(* Logix 5000 project; controller reports 1756-L63 rev 20.11; software revision 20.04; part 10 of 52 *)

        [149].log_data[0].minminute := 45, [149].log_data[0].maxminute := 45, [149].log_data[0].valid := 1, [149].log_data[1].valid := 1, [149].log_data[2].valid := 1, [149].log_data[3].valid := 1, [149].log_data[4].valid := 1, [149].log_data[5].valid := 1, [149].log_data[6].valid := 1, [149].log_data[7].valid := 1, [149].log_data[8].valid := 1, [149].log_data[9].valid := 1, [149].log_data[10].valid := 1, [149].log_data[11].valid := 1, [149].log_data[12].valid := 1, [149].log_data[13].valid := 1, [149].log_data[14].valid := 1, [149].log_data[15].valid := 1, [149].log_data[16].valid := 1, [149].log_data[17].valid := 1, [149].log_data[18].valid := 1, [149].log_data[19].valid := 1, [149].time.Year := 2023, [149].time.Month := 1, [149].time.Day := 18, [149].time.Hour := 12, [149].time.Minute := 49, [149].time.Second := 59, [150].log_data[0].min := 1.0, [150].log_data[0].max := 1.0, [150].log_data[0].total := 300.0, [150].log_data[0].time := 300.0, [150].log_data[0].minminute := 50, [150].log_data[0].maxminute := 50, [150].log_data[0].valid := 1, [150].log_data[1].valid := 1, [150].log_data[2].valid := 1, [150].log_data[3].valid := 1, [150].log_data[4].valid := 1, [150].log_data[5].valid := 1, [150].log_data[6].valid := 1, [150].log_data[7].valid := 1, [150].log_data[8].valid := 1, [150].log_data[9].valid := 1, [150].log_data[10].valid := 1, [150].log_data[11].valid := 1, [150].log_data[12].valid := 1, [150].log_data[13].valid := 1, [150].log_data[14].valid := 1, [150].log_data[15].valid := 1, [150].log_data[16].valid := 1, [150].log_data[17].valid := 1, [150].log_data[18].valid := 1, [150].log_data[19].valid := 1, [150].time.Year := 2023, [150].time.Month := 1, [150].time.Day := 18, [150].time.Hour := 12, [150].time.Minute := 54, [150].time.Second := 59,
        [151].log_data[0].min := 1.0, [151].log_data[0].max := 1.0, [151].log_data[0].total := 300.0, [151].log_data[0].time := 300.0, [151].log_data[0].minminute := 55, [151].log_data[0].maxminute := 55, [151].log_data[0].valid := 1, [151].log_data[1].valid := 1, [151].log_data[2].valid := 1, [151].log_data[3].valid := 1, [151].log_data[4].valid := 1, [151].log_data[5].valid := 1, [151].log_data[6].valid := 1, [151].log_data[7].valid := 1, [151].log_data[8].valid := 1, [151].log_data[9].valid := 1, [151].log_data[10].valid := 1, [151].log_data[11].valid := 1, [151].log_data[12].valid := 1, [151].log_data[13].valid := 1, [151].log_data[14].valid := 1, [151].log_data[15].valid := 1, [151].log_data[16].valid := 1, [151].log_data[17].valid := 1, [151].log_data[18].valid := 1, [151].log_data[19].valid := 1, [151].time.Year := 2023, [151].time.Month := 1, [151].time.Day := 18, [151].time.Hour := 12, [151].time.Minute := 59, [151].time.Second := 59, [152].log_data[0].min := 1.0, [152].log_data[0].max := 1.0, [152].log_data[0].total := 300.0, [152].log_data[0].time := 300.0, [152].log_data[0].valid := 1, [152].log_data[1].valid := 1, [152].log_data[2].valid := 1, [152].log_data[3].valid := 1, [152].log_data[4].valid := 1, [152].log_data[5].valid := 1, [152].log_data[6].valid := 1, [152].log_data[7].valid := 1, [152].log_data[8].valid := 1, [152].log_data[9].valid := 1, [152].log_data[10].valid := 1, [152].log_data[11].valid := 1, [152].log_data[12].valid := 1, [152].log_data[13].valid := 1, [152].log_data[14].valid := 1, [152].log_data[15].valid := 1, [152].log_data[16].valid := 1, [152].log_data[17].valid := 1, [152].log_data[18].valid := 1, [152].log_data[19].valid := 1, [152].time.Year := 2023, [152].time.Month := 1, [152].time.Day := 18, [152].time.Hour := 13,
        [152].time.Minute := 4, [152].time.Second := 59, [153].log_data[0].min := 1.0, [153].log_data[0].max := 1.0, [153].log_data[0].total := 300.0, [153].log_data[0].time := 300.0, [153].log_data[0].minminute := 5, [153].log_data[0].maxminute := 5, [153].log_data[0].valid := 1, [153].log_data[1].valid := 1, [153].log_data[2].valid := 1, [153].log_data[3].valid := 1, [153].log_data[4].valid := 1, [153].log_data[5].valid := 1, [153].log_data[6].valid := 1, [153].log_data[7].valid := 1, [153].log_data[8].valid := 1, [153].log_data[9].valid := 1, [153].log_data[10].valid := 1, [153].log_data[11].valid := 1, [153].log_data[12].valid := 1, [153].log_data[13].valid := 1, [153].log_data[14].valid := 1, [153].log_data[15].valid := 1, [153].log_data[16].valid := 1, [153].log_data[17].valid := 1, [153].log_data[18].valid := 1, [153].log_data[19].valid := 1, [153].time.Year := 2023, [153].time.Month := 1, [153].time.Day := 18, [153].time.Hour := 13, [153].time.Minute := 9, [153].time.Second := 59, [154].log_data[0].min := 1.0, [154].log_data[0].max := 1.0, [154].log_data[0].total := 300.0, [154].log_data[0].time := 300.0, [154].log_data[0].minminute := 10, [154].log_data[0].maxminute := 10, [154].log_data[0].valid := 1, [154].log_data[1].valid := 1, [154].log_data[2].valid := 1, [154].log_data[3].valid := 1, [154].log_data[4].valid := 1, [154].log_data[5].valid := 1, [154].log_data[6].valid := 1, [154].log_data[7].valid := 1, [154].log_data[8].valid := 1, [154].log_data[9].valid := 1, [154].log_data[10].valid := 1, [154].log_data[11].valid := 1, [154].log_data[12].valid := 1, [154].log_data[13].valid := 1, [154].log_data[14].valid := 1, [154].log_data[15].valid := 1, [154].log_data[16].valid := 1, [154].log_data[17].valid := 1, [154].log_data[18].valid := 1, [154].log_data[19].valid := 1,
        [154].time.Year := 2023, [154].time.Month := 1, [154].time.Day := 18, [154].time.Hour := 13, [154].time.Minute := 14, [154].time.Second := 59, [155].log_data[0].min := 1.0, [155].log_data[0].max := 1.0, [155].log_data[0].total := 300.0, [155].log_data[0].time := 300.0, [155].log_data[0].minminute := 15, [155].log_data[0].maxminute := 15, [155].log_data[0].valid := 1, [155].log_data[1].valid := 1, [155].log_data[2].valid := 1, [155].log_data[3].valid := 1, [155].log_data[4].valid := 1, [155].log_data[5].valid := 1, [155].log_data[6].valid := 1, [155].log_data[7].valid := 1, [155].log_data[8].valid := 1, [155].log_data[9].valid := 1, [155].log_data[10].valid := 1, [155].log_data[11].valid := 1, [155].log_data[12].valid := 1, [155].log_data[13].valid := 1, [155].log_data[14].valid := 1, [155].log_data[15].valid := 1, [155].log_data[16].valid := 1, [155].log_data[17].valid := 1, [155].log_data[18].valid := 1, [155].log_data[19].valid := 1, [155].time.Year := 2023, [155].time.Month := 1, [155].time.Day := 18, [155].time.Hour := 13, [155].time.Minute := 19, [155].time.Second := 59, [156].log_data[0].min := 1.0, [156].log_data[0].max := 1.0, [156].log_data[0].total := 300.0, [156].log_data[0].time := 300.0, [156].log_data[0].minminute := 20, [156].log_data[0].maxminute := 20, [156].log_data[0].valid := 1, [156].log_data[1].valid := 1, [156].log_data[2].valid := 1, [156].log_data[3].valid := 1, [156].log_data[4].valid := 1, [156].log_data[5].valid := 1, [156].log_data[6].valid := 1, [156].log_data[7].valid := 1, [156].log_data[8].valid := 1, [156].log_data[9].valid := 1, [156].log_data[10].valid := 1, [156].log_data[11].valid := 1, [156].log_data[12].valid := 1, [156].log_data[13].valid := 1, [156].log_data[14].valid := 1, [156].log_data[15].valid := 1,
        [156].log_data[16].valid := 1, [156].log_data[17].valid := 1, [156].log_data[18].valid := 1, [156].log_data[19].valid := 1, [156].time.Year := 2023, [156].time.Month := 1, [156].time.Day := 18, [156].time.Hour := 13, [156].time.Minute := 24, [156].time.Second := 59, [157].log_data[0].min := 1.0, [157].log_data[0].max := 1.0, [157].log_data[0].total := 300.0, [157].log_data[0].time := 300.0, [157].log_data[0].minminute := 25, [157].log_data[0].maxminute := 25, [157].log_data[0].valid := 1, [157].log_data[1].valid := 1, [157].log_data[2].valid := 1, [157].log_data[3].valid := 1, [157].log_data[4].valid := 1, [157].log_data[5].valid := 1, [157].log_data[6].valid := 1, [157].log_data[7].valid := 1, [157].log_data[8].valid := 1, [157].log_data[9].valid := 1, [157].log_data[10].valid := 1, [157].log_data[11].valid := 1, [157].log_data[12].valid := 1, [157].log_data[13].valid := 1, [157].log_data[14].valid := 1, [157].log_data[15].valid := 1, [157].log_data[16].valid := 1, [157].log_data[17].valid := 1, [157].log_data[18].valid := 1, [157].log_data[19].valid := 1, [157].time.Year := 2023, [157].time.Month := 1, [157].time.Day := 18, [157].time.Hour := 13, [157].time.Minute := 29, [157].time.Second := 59, [158].log_data[0].min := 1.0, [158].log_data[0].max := 1.0, [158].log_data[0].total := 300.0, [158].log_data[0].time := 300.0, [158].log_data[0].minminute := 30, [158].log_data[0].maxminute := 30, [158].log_data[0].valid := 1, [158].log_data[1].valid := 1, [158].log_data[2].valid := 1, [158].log_data[3].valid := 1, [158].log_data[4].valid := 1, [158].log_data[5].valid := 1, [158].log_data[6].valid := 1, [158].log_data[7].valid := 1, [158].log_data[8].valid := 1, [158].log_data[9].valid := 1, [158].log_data[10].valid := 1, [158].log_data[11].valid := 1,
        [158].log_data[12].valid := 1, [158].log_data[13].valid := 1, [158].log_data[14].valid := 1, [158].log_data[15].valid := 1, [158].log_data[16].valid := 1, [158].log_data[17].valid := 1, [158].log_data[18].valid := 1, [158].log_data[19].valid := 1, [158].time.Year := 2023, [158].time.Month := 1, [158].time.Day := 18, [158].time.Hour := 13, [158].time.Minute := 34, [158].time.Second := 59, [159].log_data[0].min := 1.0, [159].log_data[0].max := 1.0, [159].log_data[0].total := 300.0, [159].log_data[0].time := 300.0, [159].log_data[0].minminute := 35, [159].log_data[0].maxminute := 35, [159].log_data[0].valid := 1, [159].log_data[1].valid := 1, [159].log_data[2].valid := 1, [159].log_data[3].valid := 1, [159].log_data[4].valid := 1, [159].log_data[5].valid := 1, [159].log_data[6].valid := 1, [159].log_data[7].valid := 1, [159].log_data[8].valid := 1, [159].log_data[9].valid := 1, [159].log_data[10].valid := 1, [159].log_data[11].valid := 1, [159].log_data[12].valid := 1, [159].log_data[13].valid := 1, [159].log_data[14].valid := 1, [159].log_data[15].valid := 1, [159].log_data[16].valid := 1, [159].log_data[17].valid := 1, [159].log_data[18].valid := 1, [159].log_data[19].valid := 1, [159].time.Year := 2023, [159].time.Month := 1, [159].time.Day := 18, [159].time.Hour := 13, [159].time.Minute := 39, [159].time.Second := 59, [160].log_data[0].min := 1.0, [160].log_data[0].max := 1.0, [160].log_data[0].total := 300.0, [160].log_data[0].time := 300.0, [160].log_data[0].minminute := 40, [160].log_data[0].maxminute := 40, [160].log_data[0].valid := 1, [160].log_data[1].valid := 1, [160].log_data[2].valid := 1, [160].log_data[3].valid := 1, [160].log_data[4].valid := 1, [160].log_data[5].valid := 1, [160].log_data[6].valid := 1, [160].log_data[7].valid := 1,
        [160].log_data[8].valid := 1, [160].log_data[9].valid := 1, [160].log_data[10].valid := 1, [160].log_data[11].valid := 1, [160].log_data[12].valid := 1, [160].log_data[13].valid := 1, [160].log_data[14].valid := 1, [160].log_data[15].valid := 1, [160].log_data[16].valid := 1, [160].log_data[17].valid := 1, [160].log_data[18].valid := 1, [160].log_data[19].valid := 1, [160].time.Year := 2023, [160].time.Month := 1, [160].time.Day := 18, [160].time.Hour := 13, [160].time.Minute := 44, [160].time.Second := 59, [161].log_data[0].min := 1.0, [161].log_data[0].max := 1.0, [161].log_data[0].total := 300.0, [161].log_data[0].time := 300.0, [161].log_data[0].minminute := 45, [161].log_data[0].maxminute := 45, [161].log_data[0].valid := 1, [161].log_data[1].valid := 1, [161].log_data[2].valid := 1, [161].log_data[3].valid := 1, [161].log_data[4].valid := 1, [161].log_data[5].valid := 1, [161].log_data[6].valid := 1, [161].log_data[7].valid := 1, [161].log_data[8].valid := 1, [161].log_data[9].valid := 1, [161].log_data[10].valid := 1, [161].log_data[11].valid := 1, [161].log_data[12].valid := 1, [161].log_data[13].valid := 1, [161].log_data[14].valid := 1, [161].log_data[15].valid := 1, [161].log_data[16].valid := 1, [161].log_data[17].valid := 1, [161].log_data[18].valid := 1, [161].log_data[19].valid := 1, [161].time.Year := 2023, [161].time.Month := 1, [161].time.Day := 18, [161].time.Hour := 13, [161].time.Minute := 49, [161].time.Second := 59, [162].log_data[0].min := 1.0, [162].log_data[0].max := 1.0, [162].log_data[0].total := 300.0, [162].log_data[0].time := 300.0, [162].log_data[0].minminute := 50, [162].log_data[0].maxminute := 50, [162].log_data[0].valid := 1, [162].log_data[1].valid := 1, [162].log_data[2].valid := 1, [162].log_data[3].valid := 1,
        [162].log_data[4].valid := 1, [162].log_data[5].valid := 1, [162].log_data[6].valid := 1, [162].log_data[7].valid := 1, [162].log_data[8].valid := 1, [162].log_data[9].valid := 1, [162].log_data[10].valid := 1, [162].log_data[11].valid := 1, [162].log_data[12].valid := 1, [162].log_data[13].valid := 1, [162].log_data[14].valid := 1, [162].log_data[15].valid := 1, [162].log_data[16].valid := 1, [162].log_data[17].valid := 1, [162].log_data[18].valid := 1, [162].log_data[19].valid := 1, [162].time.Year := 2023, [162].time.Month := 1, [162].time.Day := 18, [162].time.Hour := 13, [162].time.Minute := 54, [162].time.Second := 59, [163].log_data[0].min := 1.0, [163].log_data[0].max := 1.0, [163].log_data[0].total := 300.0, [163].log_data[0].time := 300.0, [163].log_data[0].minminute := 55, [163].log_data[0].maxminute := 55, [163].log_data[0].valid := 1, [163].log_data[1].valid := 1, [163].log_data[2].valid := 1, [163].log_data[3].valid := 1, [163].log_data[4].valid := 1, [163].log_data[5].valid := 1, [163].log_data[6].valid := 1, [163].log_data[7].valid := 1, [163].log_data[8].valid := 1, [163].log_data[9].valid := 1, [163].log_data[10].valid := 1, [163].log_data[11].valid := 1, [163].log_data[12].valid := 1, [163].log_data[13].valid := 1, [163].log_data[14].valid := 1, [163].log_data[15].valid := 1, [163].log_data[16].valid := 1, [163].log_data[17].valid := 1, [163].log_data[18].valid := 1, [163].log_data[19].valid := 1, [163].time.Year := 2023, [163].time.Month := 1, [163].time.Day := 18, [163].time.Hour := 13, [163].time.Minute := 59, [163].time.Second := 59, [164].log_data[0].min := 1.0, [164].log_data[0].max := 1.0, [164].log_data[0].total := 300.0, [164].log_data[0].time := 300.0, [164].log_data[0].valid := 1, [164].log_data[1].valid := 1,
        [164].log_data[2].valid := 1, [164].log_data[3].valid := 1, [164].log_data[4].valid := 1, [164].log_data[5].valid := 1, [164].log_data[6].valid := 1, [164].log_data[7].valid := 1, [164].log_data[8].valid := 1, [164].log_data[9].valid := 1, [164].log_data[10].valid := 1, [164].log_data[11].valid := 1, [164].log_data[12].valid := 1, [164].log_data[13].valid := 1, [164].log_data[14].valid := 1, [164].log_data[15].valid := 1, [164].log_data[16].valid := 1, [164].log_data[17].valid := 1, [164].log_data[18].valid := 1, [164].log_data[19].valid := 1, [164].time.Year := 2023, [164].time.Month := 1, [164].time.Day := 18, [164].time.Hour := 14, [164].time.Minute := 4, [164].time.Second := 59, [165].log_data[0].min := 1.0, [165].log_data[0].max := 1.0, [165].log_data[0].total := 300.0, [165].log_data[0].time := 300.0, [165].log_data[0].minminute := 5, [165].log_data[0].maxminute := 5, [165].log_data[0].valid := 1, [165].log_data[1].valid := 1, [165].log_data[2].valid := 1, [165].log_data[3].valid := 1, [165].log_data[4].valid := 1, [165].log_data[5].valid := 1, [165].log_data[6].valid := 1, [165].log_data[7].valid := 1, [165].log_data[8].valid := 1, [165].log_data[9].valid := 1, [165].log_data[10].valid := 1, [165].log_data[11].valid := 1, [165].log_data[12].valid := 1, [165].log_data[13].valid := 1, [165].log_data[14].valid := 1, [165].log_data[15].valid := 1, [165].log_data[16].valid := 1, [165].log_data[17].valid := 1, [165].log_data[18].valid := 1, [165].log_data[19].valid := 1, [165].time.Year := 2023, [165].time.Month := 1, [165].time.Day := 18, [165].time.Hour := 14, [165].time.Minute := 9, [165].time.Second := 59, [166].log_data[0].min := 1.0, [166].log_data[0].max := 1.0, [166].log_data[0].total := 300.0, [166].log_data[0].time := 300.0,
        [166].log_data[0].minminute := 10, [166].log_data[0].maxminute := 10, [166].log_data[0].valid := 1, [166].log_data[1].valid := 1, [166].log_data[2].valid := 1, [166].log_data[3].valid := 1, [166].log_data[4].valid := 1, [166].log_data[5].valid := 1, [166].log_data[6].valid := 1, [166].log_data[7].valid := 1, [166].log_data[8].valid := 1, [166].log_data[9].valid := 1, [166].log_data[10].valid := 1, [166].log_data[11].valid := 1, [166].log_data[12].valid := 1, [166].log_data[13].valid := 1, [166].log_data[14].valid := 1, [166].log_data[15].valid := 1, [166].log_data[16].valid := 1, [166].log_data[17].valid := 1, [166].log_data[18].valid := 1, [166].log_data[19].valid := 1, [166].time.Year := 2023, [166].time.Month := 1, [166].time.Day := 18, [166].time.Hour := 14, [166].time.Minute := 14, [166].time.Second := 59, [167].log_data[0].min := 1.0, [167].log_data[0].max := 1.0, [167].log_data[0].total := 300.0, [167].log_data[0].time := 300.0, [167].log_data[0].minminute := 15, [167].log_data[0].maxminute := 15, [167].log_data[0].valid := 1, [167].log_data[1].valid := 1, [167].log_data[2].valid := 1, [167].log_data[3].valid := 1, [167].log_data[4].valid := 1, [167].log_data[5].valid := 1, [167].log_data[6].valid := 1, [167].log_data[7].valid := 1, [167].log_data[8].valid := 1, [167].log_data[9].valid := 1, [167].log_data[10].valid := 1, [167].log_data[11].valid := 1, [167].log_data[12].valid := 1, [167].log_data[13].valid := 1, [167].log_data[14].valid := 1, [167].log_data[15].valid := 1, [167].log_data[16].valid := 1, [167].log_data[17].valid := 1, [167].log_data[18].valid := 1, [167].log_data[19].valid := 1, [167].time.Year := 2023, [167].time.Month := 1, [167].time.Day := 18, [167].time.Hour := 14, [167].time.Minute := 19, [167].time.Second := 59,
        [168].log_data[0].min := 1.0, [168].log_data[0].max := 1.0, [168].log_data[0].total := 300.0, [168].log_data[0].time := 300.0, [168].log_data[0].minminute := 20, [168].log_data[0].maxminute := 20, [168].log_data[0].valid := 1, [168].log_data[1].valid := 1, [168].log_data[2].valid := 1, [168].log_data[3].valid := 1, [168].log_data[4].valid := 1, [168].log_data[5].valid := 1, [168].log_data[6].valid := 1, [168].log_data[7].valid := 1, [168].log_data[8].valid := 1, [168].log_data[9].valid := 1, [168].log_data[10].valid := 1, [168].log_data[11].valid := 1, [168].log_data[12].valid := 1, [168].log_data[13].valid := 1, [168].log_data[14].valid := 1, [168].log_data[15].valid := 1, [168].log_data[16].valid := 1, [168].log_data[17].valid := 1, [168].log_data[18].valid := 1, [168].log_data[19].valid := 1, [168].time.Year := 2023, [168].time.Month := 1, [168].time.Day := 18, [168].time.Hour := 14, [168].time.Minute := 24, [168].time.Second := 59, [169].log_data[0].min := 1.0, [169].log_data[0].max := 1.0, [169].log_data[0].total := 300.0, [169].log_data[0].time := 300.0, [169].log_data[0].minminute := 25, [169].log_data[0].maxminute := 25, [169].log_data[0].valid := 1, [169].log_data[1].valid := 1, [169].log_data[2].valid := 1, [169].log_data[3].valid := 1, [169].log_data[4].valid := 1, [169].log_data[5].valid := 1, [169].log_data[6].valid := 1, [169].log_data[7].valid := 1, [169].log_data[8].valid := 1, [169].log_data[9].valid := 1, [169].log_data[10].valid := 1, [169].log_data[11].valid := 1, [169].log_data[12].valid := 1, [169].log_data[13].valid := 1, [169].log_data[14].valid := 1, [169].log_data[15].valid := 1, [169].log_data[16].valid := 1, [169].log_data[17].valid := 1, [169].log_data[18].valid := 1, [169].log_data[19].valid := 1, [169].time.Year := 2023, [169].time.Month := 1,
        [169].time.Day := 18, [169].time.Hour := 14, [169].time.Minute := 29, [169].time.Second := 59, [170].log_data[0].min := 1.0, [170].log_data[0].max := 1.0, [170].log_data[0].total := 300.0, [170].log_data[0].time := 300.0, [170].log_data[0].minminute := 30, [170].log_data[0].maxminute := 30, [170].log_data[0].valid := 1, [170].log_data[1].valid := 1, [170].log_data[2].valid := 1, [170].log_data[3].valid := 1, [170].log_data[4].valid := 1, [170].log_data[5].valid := 1, [170].log_data[6].valid := 1, [170].log_data[7].valid := 1, [170].log_data[8].valid := 1, [170].log_data[9].valid := 1, [170].log_data[10].valid := 1, [170].log_data[11].valid := 1, [170].log_data[12].valid := 1, [170].log_data[13].valid := 1, [170].log_data[14].valid := 1, [170].log_data[15].valid := 1, [170].log_data[16].valid := 1, [170].log_data[17].valid := 1, [170].log_data[18].valid := 1, [170].log_data[19].valid := 1, [170].time.Year := 2023, [170].time.Month := 1, [170].time.Day := 18, [170].time.Hour := 14, [170].time.Minute := 34, [170].time.Second := 59, [171].log_data[0].min := 1.0, [171].log_data[0].max := 1.0, [171].log_data[0].total := 300.0, [171].log_data[0].time := 300.0, [171].log_data[0].minminute := 35, [171].log_data[0].maxminute := 35, [171].log_data[0].valid := 1, [171].log_data[1].valid := 1, [171].log_data[2].valid := 1, [171].log_data[3].valid := 1, [171].log_data[4].valid := 1, [171].log_data[5].valid := 1, [171].log_data[6].valid := 1, [171].log_data[7].valid := 1, [171].log_data[8].valid := 1, [171].log_data[9].valid := 1, [171].log_data[10].valid := 1, [171].log_data[11].valid := 1, [171].log_data[12].valid := 1, [171].log_data[13].valid := 1, [171].log_data[14].valid := 1, [171].log_data[15].valid := 1, [171].log_data[16].valid := 1, [171].log_data[17].valid := 1,
        [171].log_data[18].valid := 1, [171].log_data[19].valid := 1, [171].time.Year := 2023, [171].time.Month := 1, [171].time.Day := 18, [171].time.Hour := 14, [171].time.Minute := 39, [171].time.Second := 59, [172].log_data[0].min := 1.0, [172].log_data[0].max := 1.0, [172].log_data[0].total := 300.0, [172].log_data[0].time := 300.0, [172].log_data[0].minminute := 40, [172].log_data[0].maxminute := 40, [172].log_data[0].valid := 1, [172].log_data[1].valid := 1, [172].log_data[2].valid := 1, [172].log_data[3].valid := 1, [172].log_data[4].valid := 1, [172].log_data[5].valid := 1, [172].log_data[6].valid := 1, [172].log_data[7].valid := 1, [172].log_data[8].valid := 1, [172].log_data[9].valid := 1, [172].log_data[10].valid := 1, [172].log_data[11].valid := 1, [172].log_data[12].valid := 1, [172].log_data[13].valid := 1, [172].log_data[14].valid := 1, [172].log_data[15].valid := 1, [172].log_data[16].valid := 1, [172].log_data[17].valid := 1, [172].log_data[18].valid := 1, [172].log_data[19].valid := 1, [172].time.Year := 2023, [172].time.Month := 1, [172].time.Day := 18, [172].time.Hour := 14, [172].time.Minute := 44, [172].time.Second := 59, [173].log_data[0].min := 1.0, [173].log_data[0].max := 1.0, [173].log_data[0].total := 300.0, [173].log_data[0].time := 300.0, [173].log_data[0].minminute := 45, [173].log_data[0].maxminute := 45, [173].log_data[0].valid := 1, [173].log_data[1].valid := 1, [173].log_data[2].valid := 1, [173].log_data[3].valid := 1, [173].log_data[4].valid := 1, [173].log_data[5].valid := 1, [173].log_data[6].valid := 1, [173].log_data[7].valid := 1, [173].log_data[8].valid := 1, [173].log_data[9].valid := 1, [173].log_data[10].valid := 1, [173].log_data[11].valid := 1, [173].log_data[12].valid := 1, [173].log_data[13].valid := 1,
        [173].log_data[14].valid := 1, [173].log_data[15].valid := 1, [173].log_data[16].valid := 1, [173].log_data[17].valid := 1, [173].log_data[18].valid := 1, [173].log_data[19].valid := 1, [173].time.Year := 2023, [173].time.Month := 1, [173].time.Day := 18, [173].time.Hour := 14, [173].time.Minute := 49, [173].time.Second := 59, [174].log_data[0].min := 1.0, [174].log_data[0].max := 1.0, [174].log_data[0].total := 300.0, [174].log_data[0].time := 300.0, [174].log_data[0].minminute := 50, [174].log_data[0].maxminute := 50, [174].log_data[0].valid := 1, [174].log_data[1].valid := 1, [174].log_data[2].valid := 1, [174].log_data[3].valid := 1, [174].log_data[4].valid := 1, [174].log_data[5].valid := 1, [174].log_data[6].valid := 1, [174].log_data[7].valid := 1, [174].log_data[8].valid := 1, [174].log_data[9].valid := 1, [174].log_data[10].valid := 1, [174].log_data[11].valid := 1, [174].log_data[12].valid := 1, [174].log_data[13].valid := 1, [174].log_data[14].valid := 1, [174].log_data[15].valid := 1, [174].log_data[16].valid := 1, [174].log_data[17].valid := 1, [174].log_data[18].valid := 1, [174].log_data[19].valid := 1, [174].time.Year := 2023, [174].time.Month := 1, [174].time.Day := 18, [174].time.Hour := 14, [174].time.Minute := 54, [174].time.Second := 59, [175].log_data[0].min := 1.0, [175].log_data[0].max := 1.0, [175].log_data[0].total := 300.0, [175].log_data[0].time := 300.0, [175].log_data[0].minminute := 55, [175].log_data[0].maxminute := 55, [175].log_data[0].valid := 1, [175].log_data[1].valid := 1, [175].log_data[2].valid := 1, [175].log_data[3].valid := 1, [175].log_data[4].valid := 1, [175].log_data[5].valid := 1, [175].log_data[6].valid := 1, [175].log_data[7].valid := 1, [175].log_data[8].valid := 1, [175].log_data[9].valid := 1,
        [175].log_data[10].valid := 1, [175].log_data[11].valid := 1, [175].log_data[12].valid := 1, [175].log_data[13].valid := 1, [175].log_data[14].valid := 1, [175].log_data[15].valid := 1, [175].log_data[16].valid := 1, [175].log_data[17].valid := 1, [175].log_data[18].valid := 1, [175].log_data[19].valid := 1, [175].time.Year := 2023, [175].time.Month := 1, [175].time.Day := 18, [175].time.Hour := 14, [175].time.Minute := 59, [175].time.Second := 59, [176].log_data[0].min := 1.0, [176].log_data[0].max := 1.0, [176].log_data[0].total := 300.0, [176].log_data[0].time := 300.0, [176].log_data[0].valid := 1, [176].log_data[1].valid := 1, [176].log_data[2].valid := 1, [176].log_data[3].valid := 1, [176].log_data[4].valid := 1, [176].log_data[5].valid := 1, [176].log_data[6].valid := 1, [176].log_data[7].valid := 1, [176].log_data[8].valid := 1, [176].log_data[9].valid := 1, [176].log_data[10].valid := 1, [176].log_data[11].valid := 1, [176].log_data[12].valid := 1, [176].log_data[13].valid := 1, [176].log_data[14].valid := 1, [176].log_data[15].valid := 1, [176].log_data[16].valid := 1, [176].log_data[17].valid := 1, [176].log_data[18].valid := 1, [176].log_data[19].valid := 1, [176].time.Year := 2023, [176].time.Month := 1, [176].time.Day := 18, [176].time.Hour := 15, [176].time.Minute := 4, [176].time.Second := 59, [177].log_data[0].min := 1.0, [177].log_data[0].max := 1.0, [177].log_data[0].total := 300.0, [177].log_data[0].time := 300.0, [177].log_data[0].minminute := 5, [177].log_data[0].maxminute := 5, [177].log_data[0].valid := 1, [177].log_data[1].valid := 1, [177].log_data[2].valid := 1, [177].log_data[3].valid := 1, [177].log_data[4].valid := 1, [177].log_data[5].valid := 1, [177].log_data[6].valid := 1, [177].log_data[7].valid := 1,
        [177].log_data[8].valid := 1, [177].log_data[9].valid := 1, [177].log_data[10].valid := 1, [177].log_data[11].valid := 1, [177].log_data[12].valid := 1, [177].log_data[13].valid := 1, [177].log_data[14].valid := 1, [177].log_data[15].valid := 1, [177].log_data[16].valid := 1, [177].log_data[17].valid := 1, [177].log_data[18].valid := 1, [177].log_data[19].valid := 1, [177].time.Year := 2023, [177].time.Month := 1, [177].time.Day := 18, [177].time.Hour := 15, [177].time.Minute := 9, [177].time.Second := 59, [178].log_data[0].min := 1.0, [178].log_data[0].max := 1.0, [178].log_data[0].total := 300.0, [178].log_data[0].time := 300.0, [178].log_data[0].minminute := 10, [178].log_data[0].maxminute := 10, [178].log_data[0].valid := 1, [178].log_data[1].valid := 1, [178].log_data[2].valid := 1, [178].log_data[3].valid := 1, [178].log_data[4].valid := 1, [178].log_data[5].valid := 1, [178].log_data[6].valid := 1, [178].log_data[7].valid := 1, [178].log_data[8].valid := 1, [178].log_data[9].valid := 1, [178].log_data[10].valid := 1, [178].log_data[11].valid := 1, [178].log_data[12].valid := 1, [178].log_data[13].valid := 1, [178].log_data[14].valid := 1, [178].log_data[15].valid := 1, [178].log_data[16].valid := 1, [178].log_data[17].valid := 1, [178].log_data[18].valid := 1, [178].log_data[19].valid := 1, [178].time.Year := 2023, [178].time.Month := 1, [178].time.Day := 18, [178].time.Hour := 15, [178].time.Minute := 14, [178].time.Second := 59, [179].log_data[0].min := 1.0, [179].log_data[0].max := 1.0, [179].log_data[0].total := 300.0, [179].log_data[0].time := 300.0, [179].log_data[0].minminute := 15, [179].log_data[0].maxminute := 15, [179].log_data[0].valid := 1, [179].log_data[1].valid := 1, [179].log_data[2].valid := 1, [179].log_data[3].valid := 1,
        [179].log_data[4].valid := 1, [179].log_data[5].valid := 1, [179].log_data[6].valid := 1, [179].log_data[7].valid := 1, [179].log_data[8].valid := 1, [179].log_data[9].valid := 1, [179].log_data[10].valid := 1, [179].log_data[11].valid := 1, [179].log_data[12].valid := 1, [179].log_data[13].valid := 1, [179].log_data[14].valid := 1, [179].log_data[15].valid := 1, [179].log_data[16].valid := 1, [179].log_data[17].valid := 1, [179].log_data[18].valid := 1, [179].log_data[19].valid := 1, [179].time.Year := 2023, [179].time.Month := 1, [179].time.Day := 18, [179].time.Hour := 15, [179].time.Minute := 19, [179].time.Second := 59, [180].log_data[0].min := 1.0, [180].log_data[0].max := 1.0, [180].log_data[0].total := 300.0, [180].log_data[0].time := 300.0, [180].log_data[0].minminute := 20, [180].log_data[0].maxminute := 20, [180].log_data[0].valid := 1, [180].log_data[1].valid := 1, [180].log_data[2].valid := 1, [180].log_data[3].valid := 1, [180].log_data[4].valid := 1, [180].log_data[5].valid := 1, [180].log_data[6].valid := 1, [180].log_data[7].valid := 1, [180].log_data[8].valid := 1, [180].log_data[9].valid := 1, [180].log_data[10].valid := 1, [180].log_data[11].valid := 1, [180].log_data[12].valid := 1, [180].log_data[13].valid := 1, [180].log_data[14].valid := 1, [180].log_data[15].valid := 1, [180].log_data[16].valid := 1, [180].log_data[17].valid := 1, [180].log_data[18].valid := 1, [180].log_data[19].valid := 1, [180].time.Year := 2023, [180].time.Month := 1, [180].time.Day := 18, [180].time.Hour := 15, [180].time.Minute := 24, [180].time.Second := 59, [181].log_data[0].min := 1.0, [181].log_data[0].max := 1.0, [181].log_data[0].total := 300.0, [181].log_data[0].time := 300.0, [181].log_data[0].minminute := 25, [181].log_data[0].maxminute := 25,
        [181].log_data[0].valid := 1, [181].log_data[1].valid := 1, [181].log_data[2].valid := 1, [181].log_data[3].valid := 1, [181].log_data[4].valid := 1, [181].log_data[5].valid := 1, [181].log_data[6].valid := 1, [181].log_data[7].valid := 1, [181].log_data[8].valid := 1, [181].log_data[9].valid := 1, [181].log_data[10].valid := 1, [181].log_data[11].valid := 1, [181].log_data[12].valid := 1, [181].log_data[13].valid := 1, [181].log_data[14].valid := 1, [181].log_data[15].valid := 1, [181].log_data[16].valid := 1, [181].log_data[17].valid := 1, [181].log_data[18].valid := 1, [181].log_data[19].valid := 1, [181].time.Year := 2023, [181].time.Month := 1, [181].time.Day := 18, [181].time.Hour := 15, [181].time.Minute := 29, [181].time.Second := 59, [182].log_data[0].min := 1.0, [182].log_data[0].max := 1.0, [182].log_data[0].total := 300.0, [182].log_data[0].time := 300.0, [182].log_data[0].minminute := 30, [182].log_data[0].maxminute := 30, [182].log_data[0].valid := 1, [182].log_data[1].valid := 1, [182].log_data[2].valid := 1, [182].log_data[3].valid := 1, [182].log_data[4].valid := 1, [182].log_data[5].valid := 1, [182].log_data[6].valid := 1, [182].log_data[7].valid := 1, [182].log_data[8].valid := 1, [182].log_data[9].valid := 1, [182].log_data[10].valid := 1, [182].log_data[11].valid := 1, [182].log_data[12].valid := 1, [182].log_data[13].valid := 1, [182].log_data[14].valid := 1, [182].log_data[15].valid := 1, [182].log_data[16].valid := 1, [182].log_data[17].valid := 1, [182].log_data[18].valid := 1, [182].log_data[19].valid := 1, [182].time.Year := 2023, [182].time.Month := 1, [182].time.Day := 18, [182].time.Hour := 15, [182].time.Minute := 34, [182].time.Second := 59, [183].log_data[0].min := 1.0, [183].log_data[0].max := 1.0,
        [183].log_data[0].total := 300.0, [183].log_data[0].time := 300.0, [183].log_data[0].minminute := 35, [183].log_data[0].maxminute := 35, [183].log_data[0].valid := 1, [183].log_data[1].valid := 1, [183].log_data[2].valid := 1, [183].log_data[3].valid := 1, [183].log_data[4].valid := 1, [183].log_data[5].valid := 1, [183].log_data[6].valid := 1, [183].log_data[7].valid := 1, [183].log_data[8].valid := 1, [183].log_data[9].valid := 1, [183].log_data[10].valid := 1, [183].log_data[11].valid := 1, [183].log_data[12].valid := 1, [183].log_data[13].valid := 1, [183].log_data[14].valid := 1, [183].log_data[15].valid := 1, [183].log_data[16].valid := 1, [183].log_data[17].valid := 1, [183].log_data[18].valid := 1, [183].log_data[19].valid := 1, [183].time.Year := 2023, [183].time.Month := 1, [183].time.Day := 18, [183].time.Hour := 15, [183].time.Minute := 39, [183].time.Second := 59, [184].log_data[0].min := 1.0, [184].log_data[0].max := 1.0, [184].log_data[0].total := 300.0, [184].log_data[0].time := 300.0, [184].log_data[0].minminute := 40, [184].log_data[0].maxminute := 40, [184].log_data[0].valid := 1, [184].log_data[1].valid := 1, [184].log_data[2].valid := 1, [184].log_data[3].valid := 1, [184].log_data[4].valid := 1, [184].log_data[5].valid := 1, [184].log_data[6].valid := 1, [184].log_data[7].valid := 1, [184].log_data[8].valid := 1, [184].log_data[9].valid := 1, [184].log_data[10].valid := 1, [184].log_data[11].valid := 1, [184].log_data[12].valid := 1, [184].log_data[13].valid := 1, [184].log_data[14].valid := 1, [184].log_data[15].valid := 1, [184].log_data[16].valid := 1, [184].log_data[17].valid := 1, [184].log_data[18].valid := 1, [184].log_data[19].valid := 1, [184].time.Year := 2023, [184].time.Month := 1, [184].time.Day := 18, [184].time.Hour := 15,
        [184].time.Minute := 44, [184].time.Second := 59, [185].log_data[0].min := 1.0, [185].log_data[0].max := 1.0, [185].log_data[0].total := 300.0, [185].log_data[0].time := 300.0, [185].log_data[0].minminute := 45, [185].log_data[0].maxminute := 45, [185].log_data[0].valid := 1, [185].log_data[1].valid := 1, [185].log_data[2].valid := 1, [185].log_data[3].valid := 1, [185].log_data[4].valid := 1, [185].log_data[5].valid := 1, [185].log_data[6].valid := 1, [185].log_data[7].valid := 1, [185].log_data[8].valid := 1, [185].log_data[9].valid := 1, [185].log_data[10].valid := 1, [185].log_data[11].valid := 1, [185].log_data[12].valid := 1, [185].log_data[13].valid := 1, [185].log_data[14].valid := 1, [185].log_data[15].valid := 1, [185].log_data[16].valid := 1, [185].log_data[17].valid := 1, [185].log_data[18].valid := 1, [185].log_data[19].valid := 1, [185].time.Year := 2023, [185].time.Month := 1, [185].time.Day := 18, [185].time.Hour := 15, [185].time.Minute := 49, [185].time.Second := 59, [186].log_data[0].min := 1.0, [186].log_data[0].max := 1.0, [186].log_data[0].total := 300.0, [186].log_data[0].time := 300.0, [186].log_data[0].minminute := 50, [186].log_data[0].maxminute := 50, [186].log_data[0].valid := 1, [186].log_data[1].valid := 1, [186].log_data[2].valid := 1, [186].log_data[3].valid := 1, [186].log_data[4].valid := 1, [186].log_data[5].valid := 1, [186].log_data[6].valid := 1, [186].log_data[7].valid := 1, [186].log_data[8].valid := 1, [186].log_data[9].valid := 1, [186].log_data[10].valid := 1, [186].log_data[11].valid := 1, [186].log_data[12].valid := 1, [186].log_data[13].valid := 1, [186].log_data[14].valid := 1, [186].log_data[15].valid := 1, [186].log_data[16].valid := 1, [186].log_data[17].valid := 1, [186].log_data[18].valid := 1, [186].log_data[19].valid := 1,
        [186].time.Year := 2023, [186].time.Month := 1, [186].time.Day := 18, [186].time.Hour := 15, [186].time.Minute := 54, [186].time.Second := 59, [187].log_data[0].min := 1.0, [187].log_data[0].max := 1.0, [187].log_data[0].total := 300.0, [187].log_data[0].time := 300.0, [187].log_data[0].minminute := 55, [187].log_data[0].maxminute := 55, [187].log_data[0].valid := 1, [187].log_data[1].valid := 1, [187].log_data[2].valid := 1, [187].log_data[3].valid := 1, [187].log_data[4].valid := 1, [187].log_data[5].valid := 1, [187].log_data[6].valid := 1, [187].log_data[7].valid := 1, [187].log_data[8].valid := 1, [187].log_data[9].valid := 1, [187].log_data[10].valid := 1, [187].log_data[11].valid := 1, [187].log_data[12].valid := 1, [187].log_data[13].valid := 1, [187].log_data[14].valid := 1, [187].log_data[15].valid := 1, [187].log_data[16].valid := 1, [187].log_data[17].valid := 1, [187].log_data[18].valid := 1, [187].log_data[19].valid := 1, [187].time.Year := 2023, [187].time.Month := 1, [187].time.Day := 18, [187].time.Hour := 15, [187].time.Minute := 59, [187].time.Second := 59, [188].log_data[0].min := 1.0, [188].log_data[0].max := 1.0, [188].log_data[0].total := 300.0, [188].log_data[0].time := 300.0, [188].log_data[0].valid := 1, [188].log_data[1].valid := 1, [188].log_data[2].valid := 1, [188].log_data[3].valid := 1, [188].log_data[4].valid := 1, [188].log_data[5].valid := 1, [188].log_data[6].valid := 1, [188].log_data[7].valid := 1, [188].log_data[8].valid := 1, [188].log_data[9].valid := 1, [188].log_data[10].valid := 1, [188].log_data[11].valid := 1, [188].log_data[12].valid := 1, [188].log_data[13].valid := 1, [188].log_data[14].valid := 1, [188].log_data[15].valid := 1, [188].log_data[16].valid := 1, [188].log_data[17].valid := 1,
        [188].log_data[18].valid := 1, [188].log_data[19].valid := 1, [188].time.Year := 2023, [188].time.Month := 1, [188].time.Day := 18, [188].time.Hour := 16, [188].time.Minute := 4, [188].time.Second := 59, [189].log_data[0].min := 1.0, [189].log_data[0].max := 1.0, [189].log_data[0].total := 300.0, [189].log_data[0].time := 300.0, [189].log_data[0].minminute := 5, [189].log_data[0].maxminute := 5, [189].log_data[0].valid := 1, [189].log_data[1].valid := 1, [189].log_data[2].valid := 1, [189].log_data[3].valid := 1, [189].log_data[4].valid := 1, [189].log_data[5].valid := 1, [189].log_data[6].valid := 1, [189].log_data[7].valid := 1, [189].log_data[8].valid := 1, [189].log_data[9].valid := 1, [189].log_data[10].valid := 1, [189].log_data[11].valid := 1, [189].log_data[12].valid := 1, [189].log_data[13].valid := 1, [189].log_data[14].valid := 1, [189].log_data[15].valid := 1, [189].log_data[16].valid := 1, [189].log_data[17].valid := 1, [189].log_data[18].valid := 1, [189].log_data[19].valid := 1, [189].time.Year := 2023, [189].time.Month := 1, [189].time.Day := 18, [189].time.Hour := 16, [189].time.Minute := 9, [189].time.Second := 59, [190].log_data[0].min := 1.0, [190].log_data[0].max := 1.0, [190].log_data[0].total := 300.0, [190].log_data[0].time := 300.0, [190].log_data[0].minminute := 10, [190].log_data[0].maxminute := 10, [190].log_data[0].valid := 1, [190].log_data[1].valid := 1, [190].log_data[2].valid := 1, [190].log_data[3].valid := 1, [190].log_data[4].valid := 1, [190].log_data[5].valid := 1, [190].log_data[6].valid := 1, [190].log_data[7].valid := 1, [190].log_data[8].valid := 1, [190].log_data[9].valid := 1, [190].log_data[10].valid := 1, [190].log_data[11].valid := 1, [190].log_data[12].valid := 1, [190].log_data[13].valid := 1,
        [190].log_data[14].valid := 1, [190].log_data[15].valid := 1, [190].log_data[16].valid := 1, [190].log_data[17].valid := 1, [190].log_data[18].valid := 1, [190].log_data[19].valid := 1, [190].time.Year := 2023, [190].time.Month := 1, [190].time.Day := 18, [190].time.Hour := 16, [190].time.Minute := 14, [190].time.Second := 59, [191].log_data[0].min := 1.0, [191].log_data[0].max := 1.0, [191].log_data[0].total := 300.0, [191].log_data[0].time := 300.0, [191].log_data[0].minminute := 15, [191].log_data[0].maxminute := 15, [191].log_data[0].valid := 1, [191].log_data[1].valid := 1, [191].log_data[2].valid := 1, [191].log_data[3].valid := 1, [191].log_data[4].valid := 1, [191].log_data[5].valid := 1, [191].log_data[6].valid := 1, [191].log_data[7].valid := 1, [191].log_data[8].valid := 1, [191].log_data[9].valid := 1, [191].log_data[10].valid := 1, [191].log_data[11].valid := 1, [191].log_data[12].valid := 1, [191].log_data[13].valid := 1, [191].log_data[14].valid := 1, [191].log_data[15].valid := 1, [191].log_data[16].valid := 1, [191].log_data[17].valid := 1, [191].log_data[18].valid := 1, [191].log_data[19].valid := 1, [191].time.Year := 2023, [191].time.Month := 1, [191].time.Day := 18, [191].time.Hour := 16, [191].time.Minute := 19, [191].time.Second := 59, [192].log_data[0].min := 1.0, [192].log_data[0].max := 1.0, [192].log_data[0].total := 300.0, [192].log_data[0].time := 300.0, [192].log_data[0].minminute := 20, [192].log_data[0].maxminute := 20, [192].log_data[0].valid := 1, [192].log_data[1].valid := 1, [192].log_data[2].valid := 1, [192].log_data[3].valid := 1, [192].log_data[4].valid := 1, [192].log_data[5].valid := 1, [192].log_data[6].valid := 1, [192].log_data[7].valid := 1, [192].log_data[8].valid := 1, [192].log_data[9].valid := 1,
        [192].log_data[10].valid := 1, [192].log_data[11].valid := 1, [192].log_data[12].valid := 1, [192].log_data[13].valid := 1, [192].log_data[14].valid := 1, [192].log_data[15].valid := 1, [192].log_data[16].valid := 1, [192].log_data[17].valid := 1, [192].log_data[18].valid := 1, [192].log_data[19].valid := 1, [192].time.Year := 2023, [192].time.Month := 1, [192].time.Day := 18, [192].time.Hour := 16, [192].time.Minute := 24, [192].time.Second := 59, [193].log_data[0].min := 1.0, [193].log_data[0].max := 1.0, [193].log_data[0].total := 300.0, [193].log_data[0].time := 300.0, [193].log_data[0].minminute := 25, [193].log_data[0].maxminute := 25, [193].log_data[0].valid := 1, [193].log_data[1].valid := 1, [193].log_data[2].valid := 1, [193].log_data[3].valid := 1, [193].log_data[4].valid := 1, [193].log_data[5].valid := 1, [193].log_data[6].valid := 1, [193].log_data[7].valid := 1, [193].log_data[8].valid := 1, [193].log_data[9].valid := 1, [193].log_data[10].valid := 1, [193].log_data[11].valid := 1, [193].log_data[12].valid := 1, [193].log_data[13].valid := 1, [193].log_data[14].valid := 1, [193].log_data[15].valid := 1, [193].log_data[16].valid := 1, [193].log_data[17].valid := 1, [193].log_data[18].valid := 1, [193].log_data[19].valid := 1, [193].time.Year := 2023, [193].time.Month := 1, [193].time.Day := 18, [193].time.Hour := 16, [193].time.Minute := 29, [193].time.Second := 59, [194].log_data[0].min := 1.0, [194].log_data[0].max := 1.0, [194].log_data[0].total := 300.0, [194].log_data[0].time := 300.0, [194].log_data[0].minminute := 30, [194].log_data[0].maxminute := 30, [194].log_data[0].valid := 1, [194].log_data[1].valid := 1, [194].log_data[2].valid := 1, [194].log_data[3].valid := 1, [194].log_data[4].valid := 1, [194].log_data[5].valid := 1,
        [194].log_data[6].valid := 1, [194].log_data[7].valid := 1, [194].log_data[8].valid := 1, [194].log_data[9].valid := 1, [194].log_data[10].valid := 1, [194].log_data[11].valid := 1, [194].log_data[12].valid := 1, [194].log_data[13].valid := 1, [194].log_data[14].valid := 1, [194].log_data[15].valid := 1, [194].log_data[16].valid := 1, [194].log_data[17].valid := 1, [194].log_data[18].valid := 1, [194].log_data[19].valid := 1, [194].time.Year := 2023, [194].time.Month := 1, [194].time.Day := 18, [194].time.Hour := 16, [194].time.Minute := 34, [194].time.Second := 59, [195].log_data[0].min := 1.0, [195].log_data[0].max := 1.0, [195].log_data[0].total := 300.0, [195].log_data[0].time := 300.0, [195].log_data[0].minminute := 35, [195].log_data[0].maxminute := 35, [195].log_data[0].valid := 1, [195].log_data[1].valid := 1, [195].log_data[2].valid := 1, [195].log_data[3].valid := 1, [195].log_data[4].valid := 1, [195].log_data[5].valid := 1, [195].log_data[6].valid := 1, [195].log_data[7].valid := 1, [195].log_data[8].valid := 1, [195].log_data[9].valid := 1, [195].log_data[10].valid := 1, [195].log_data[11].valid := 1, [195].log_data[12].valid := 1, [195].log_data[13].valid := 1, [195].log_data[14].valid := 1, [195].log_data[15].valid := 1, [195].log_data[16].valid := 1, [195].log_data[17].valid := 1, [195].log_data[18].valid := 1, [195].log_data[19].valid := 1, [195].time.Year := 2023, [195].time.Month := 1, [195].time.Day := 18, [195].time.Hour := 16, [195].time.Minute := 39, [195].time.Second := 59, [196].log_data[0].min := 1.0, [196].log_data[0].max := 1.0, [196].log_data[0].total := 300.0, [196].log_data[0].time := 300.0, [196].log_data[0].minminute := 40, [196].log_data[0].maxminute := 40, [196].log_data[0].valid := 1, [196].log_data[1].valid := 1,
        [196].log_data[2].valid := 1, [196].log_data[3].valid := 1, [196].log_data[4].valid := 1, [196].log_data[5].valid := 1, [196].log_data[6].valid := 1, [196].log_data[7].valid := 1, [196].log_data[8].valid := 1, [196].log_data[9].valid := 1, [196].log_data[10].valid := 1, [196].log_data[11].valid := 1, [196].log_data[12].valid := 1, [196].log_data[13].valid := 1, [196].log_data[14].valid := 1, [196].log_data[15].valid := 1, [196].log_data[16].valid := 1, [196].log_data[17].valid := 1, [196].log_data[18].valid := 1, [196].log_data[19].valid := 1, [196].time.Year := 2023, [196].time.Month := 1, [196].time.Day := 18, [196].time.Hour := 16, [196].time.Minute := 44, [196].time.Second := 59, [197].log_data[0].min := 1.0, [197].log_data[0].max := 1.0, [197].log_data[0].total := 300.0, [197].log_data[0].time := 300.0, [197].log_data[0].minminute := 45, [197].log_data[0].maxminute := 45, [197].log_data[0].valid := 1, [197].log_data[1].valid := 1, [197].log_data[2].valid := 1, [197].log_data[3].valid := 1, [197].log_data[4].valid := 1, [197].log_data[5].valid := 1, [197].log_data[6].valid := 1, [197].log_data[7].valid := 1, [197].log_data[8].valid := 1, [197].log_data[9].valid := 1, [197].log_data[10].valid := 1, [197].log_data[11].valid := 1, [197].log_data[12].valid := 1, [197].log_data[13].valid := 1, [197].log_data[14].valid := 1, [197].log_data[15].valid := 1, [197].log_data[16].valid := 1, [197].log_data[17].valid := 1, [197].log_data[18].valid := 1, [197].log_data[19].valid := 1, [197].time.Year := 2023, [197].time.Month := 1, [197].time.Day := 18, [197].time.Hour := 16, [197].time.Minute := 49, [197].time.Second := 59, [198].log_data[0].min := 1.0, [198].log_data[0].max := 1.0, [198].log_data[0].total := 300.0, [198].log_data[0].time := 300.0,
        [198].log_data[0].minminute := 50, [198].log_data[0].maxminute := 50, [198].log_data[0].valid := 1, [198].log_data[1].valid := 1, [198].log_data[2].valid := 1, [198].log_data[3].valid := 1, [198].log_data[4].valid := 1, [198].log_data[5].valid := 1, [198].log_data[6].valid := 1, [198].log_data[7].valid := 1, [198].log_data[8].valid := 1, [198].log_data[9].valid := 1, [198].log_data[10].valid := 1, [198].log_data[11].valid := 1, [198].log_data[12].valid := 1, [198].log_data[13].valid := 1, [198].log_data[14].valid := 1, [198].log_data[15].valid := 1, [198].log_data[16].valid := 1, [198].log_data[17].valid := 1, [198].log_data[18].valid := 1, [198].log_data[19].valid := 1, [198].time.Year := 2023, [198].time.Month := 1, [198].time.Day := 18, [198].time.Hour := 16, [198].time.Minute := 54, [198].time.Second := 59, [199].log_data[0].min := 1.0, [199].log_data[0].max := 1.0, [199].log_data[0].total := 300.0, [199].log_data[0].time := 300.0, [199].log_data[0].minminute := 55, [199].log_data[0].maxminute := 55, [199].log_data[0].valid := 1, [199].log_data[1].valid := 1, [199].log_data[2].valid := 1, [199].log_data[3].valid := 1, [199].log_data[4].valid := 1, [199].log_data[5].valid := 1, [199].log_data[6].valid := 1, [199].log_data[7].valid := 1, [199].log_data[8].valid := 1, [199].log_data[9].valid := 1, [199].log_data[10].valid := 1, [199].log_data[11].valid := 1, [199].log_data[12].valid := 1, [199].log_data[13].valid := 1, [199].log_data[14].valid := 1, [199].log_data[15].valid := 1, [199].log_data[16].valid := 1, [199].log_data[17].valid := 1, [199].log_data[18].valid := 1, [199].log_data[19].valid := 1, [199].time.Year := 2023, [199].time.Month := 1, [199].time.Day := 18, [199].time.Hour := 16, [199].time.Minute := 59, [199].time.Second := 59,
        [200].log_data[0].min := 1.0, [200].log_data[0].max := 1.0, [200].log_data[0].total := 300.0, [200].log_data[0].time := 300.0, [200].log_data[0].valid := 1, [200].log_data[1].valid := 1, [200].log_data[2].valid := 1, [200].log_data[3].valid := 1, [200].log_data[4].valid := 1, [200].log_data[5].valid := 1, [200].log_data[6].valid := 1, [200].log_data[7].valid := 1, [200].log_data[8].valid := 1, [200].log_data[9].valid := 1, [200].log_data[10].valid := 1, [200].log_data[11].valid := 1, [200].log_data[12].valid := 1, [200].log_data[13].valid := 1, [200].log_data[14].valid := 1, [200].log_data[15].valid := 1, [200].log_data[16].valid := 1, [200].log_data[17].valid := 1, [200].log_data[18].valid := 1, [200].log_data[19].valid := 1, [200].time.Year := 2023, [200].time.Month := 1, [200].time.Day := 18, [200].time.Hour := 17, [200].time.Minute := 4, [200].time.Second := 59, [201].log_data[0].min := 1.0, [201].log_data[0].max := 1.0, [201].log_data[0].total := 300.0, [201].log_data[0].time := 300.0, [201].log_data[0].minminute := 5, [201].log_data[0].maxminute := 5, [201].log_data[0].valid := 1, [201].log_data[1].valid := 1, [201].log_data[2].valid := 1, [201].log_data[3].valid := 1, [201].log_data[4].valid := 1, [201].log_data[5].valid := 1, [201].log_data[6].valid := 1, [201].log_data[7].valid := 1, [201].log_data[8].valid := 1, [201].log_data[9].valid := 1, [201].log_data[10].valid := 1, [201].log_data[11].valid := 1, [201].log_data[12].valid := 1, [201].log_data[13].valid := 1, [201].log_data[14].valid := 1, [201].log_data[15].valid := 1, [201].log_data[16].valid := 1, [201].log_data[17].valid := 1, [201].log_data[18].valid := 1, [201].log_data[19].valid := 1, [201].time.Year := 2023, [201].time.Month := 1, [201].time.Day := 18, [201].time.Hour := 17,
        [201].time.Minute := 9, [201].time.Second := 59, [202].log_data[0].min := 1.0, [202].log_data[0].max := 1.0, [202].log_data[0].total := 300.0, [202].log_data[0].time := 300.0, [202].log_data[0].minminute := 10, [202].log_data[0].maxminute := 10, [202].log_data[0].valid := 1, [202].log_data[1].valid := 1, [202].log_data[2].valid := 1, [202].log_data[3].valid := 1, [202].log_data[4].valid := 1, [202].log_data[5].valid := 1, [202].log_data[6].valid := 1, [202].log_data[7].valid := 1, [202].log_data[8].valid := 1, [202].log_data[9].valid := 1, [202].log_data[10].valid := 1, [202].log_data[11].valid := 1, [202].log_data[12].valid := 1, [202].log_data[13].valid := 1, [202].log_data[14].valid := 1, [202].log_data[15].valid := 1, [202].log_data[16].valid := 1, [202].log_data[17].valid := 1, [202].log_data[18].valid := 1, [202].log_data[19].valid := 1, [202].time.Year := 2023, [202].time.Month := 1, [202].time.Day := 18, [202].time.Hour := 17, [202].time.Minute := 14, [202].time.Second := 59, [203].log_data[0].min := 1.0, [203].log_data[0].max := 1.0, [203].log_data[0].total := 300.0, [203].log_data[0].time := 300.0, [203].log_data[0].minminute := 15, [203].log_data[0].maxminute := 15, [203].log_data[0].valid := 1, [203].log_data[1].valid := 1, [203].log_data[2].valid := 1, [203].log_data[3].valid := 1, [203].log_data[4].valid := 1, [203].log_data[5].valid := 1, [203].log_data[6].valid := 1, [203].log_data[7].valid := 1, [203].log_data[8].valid := 1, [203].log_data[9].valid := 1, [203].log_data[10].valid := 1, [203].log_data[11].valid := 1, [203].log_data[12].valid := 1, [203].log_data[13].valid := 1, [203].log_data[14].valid := 1, [203].log_data[15].valid := 1, [203].log_data[16].valid := 1, [203].log_data[17].valid := 1, [203].log_data[18].valid := 1, [203].log_data[19].valid := 1,
        [203].time.Year := 2023, [203].time.Month := 1, [203].time.Day := 18, [203].time.Hour := 17, [203].time.Minute := 19, [203].time.Second := 59, [204].log_data[0].min := 1.0, [204].log_data[0].max := 1.0, [204].log_data[0].total := 300.0, [204].log_data[0].time := 300.0, [204].log_data[0].minminute := 20, [204].log_data[0].maxminute := 20, [204].log_data[0].valid := 1, [204].log_data[1].valid := 1, [204].log_data[2].valid := 1, [204].log_data[3].valid := 1, [204].log_data[4].valid := 1, [204].log_data[5].valid := 1, [204].log_data[6].valid := 1, [204].log_data[7].valid := 1, [204].log_data[8].valid := 1, [204].log_data[9].valid := 1, [204].log_data[10].valid := 1, [204].log_data[11].valid := 1, [204].log_data[12].valid := 1, [204].log_data[13].valid := 1, [204].log_data[14].valid := 1, [204].log_data[15].valid := 1, [204].log_data[16].valid := 1, [204].log_data[17].valid := 1, [204].log_data[18].valid := 1, [204].log_data[19].valid := 1, [204].time.Year := 2023, [204].time.Month := 1, [204].time.Day := 18, [204].time.Hour := 17, [204].time.Minute := 24, [204].time.Second := 59, [205].log_data[0].min := 1.0, [205].log_data[0].max := 1.0, [205].log_data[0].total := 300.0, [205].log_data[0].time := 300.0, [205].log_data[0].minminute := 25, [205].log_data[0].maxminute := 25, [205].log_data[0].valid := 1, [205].log_data[1].valid := 1, [205].log_data[2].valid := 1, [205].log_data[3].valid := 1, [205].log_data[4].valid := 1, [205].log_data[5].valid := 1, [205].log_data[6].valid := 1, [205].log_data[7].valid := 1, [205].log_data[8].valid := 1, [205].log_data[9].valid := 1, [205].log_data[10].valid := 1, [205].log_data[11].valid := 1, [205].log_data[12].valid := 1, [205].log_data[13].valid := 1, [205].log_data[14].valid := 1, [205].log_data[15].valid := 1,
        [205].log_data[16].valid := 1, [205].log_data[17].valid := 1, [205].log_data[18].valid := 1, [205].log_data[19].valid := 1, [205].time.Year := 2023, [205].time.Month := 1, [205].time.Day := 18, [205].time.Hour := 17, [205].time.Minute := 29, [205].time.Second := 59, [206].log_data[0].min := 1.0, [206].log_data[0].max := 1.0, [206].log_data[0].total := 300.0, [206].log_data[0].time := 300.0, [206].log_data[0].minminute := 30, [206].log_data[0].maxminute := 30, [206].log_data[0].valid := 1, [206].log_data[1].valid := 1, [206].log_data[2].valid := 1, [206].log_data[3].valid := 1, [206].log_data[4].valid := 1, [206].log_data[5].valid := 1, [206].log_data[6].valid := 1, [206].log_data[7].valid := 1, [206].log_data[8].valid := 1, [206].log_data[9].valid := 1, [206].log_data[10].valid := 1, [206].log_data[11].valid := 1, [206].log_data[12].valid := 1, [206].log_data[13].valid := 1, [206].log_data[14].valid := 1, [206].log_data[15].valid := 1, [206].log_data[16].valid := 1, [206].log_data[17].valid := 1, [206].log_data[18].valid := 1, [206].log_data[19].valid := 1, [206].time.Year := 2023, [206].time.Month := 1, [206].time.Day := 18, [206].time.Hour := 17, [206].time.Minute := 34, [206].time.Second := 59, [207].log_data[0].min := 1.0, [207].log_data[0].max := 1.0, [207].log_data[0].total := 300.0, [207].log_data[0].time := 300.0, [207].log_data[0].minminute := 35, [207].log_data[0].maxminute := 35, [207].log_data[0].valid := 1, [207].log_data[1].valid := 1, [207].log_data[2].valid := 1, [207].log_data[3].valid := 1, [207].log_data[4].valid := 1, [207].log_data[5].valid := 1, [207].log_data[6].valid := 1, [207].log_data[7].valid := 1, [207].log_data[8].valid := 1, [207].log_data[9].valid := 1, [207].log_data[10].valid := 1, [207].log_data[11].valid := 1,
        [207].log_data[12].valid := 1, [207].log_data[13].valid := 1, [207].log_data[14].valid := 1, [207].log_data[15].valid := 1, [207].log_data[16].valid := 1, [207].log_data[17].valid := 1, [207].log_data[18].valid := 1, [207].log_data[19].valid := 1, [207].time.Year := 2023, [207].time.Month := 1, [207].time.Day := 18, [207].time.Hour := 17, [207].time.Minute := 39, [207].time.Second := 59, [208].log_data[0].min := 1.0, [208].log_data[0].max := 1.0, [208].log_data[0].total := 300.0, [208].log_data[0].time := 300.0, [208].log_data[0].minminute := 40, [208].log_data[0].maxminute := 40, [208].log_data[0].valid := 1, [208].log_data[1].valid := 1, [208].log_data[2].valid := 1, [208].log_data[3].valid := 1, [208].log_data[4].valid := 1, [208].log_data[5].valid := 1, [208].log_data[6].valid := 1, [208].log_data[7].valid := 1, [208].log_data[8].valid := 1, [208].log_data[9].valid := 1, [208].log_data[10].valid := 1, [208].log_data[11].valid := 1, [208].log_data[12].valid := 1, [208].log_data[13].valid := 1, [208].log_data[14].valid := 1, [208].log_data[15].valid := 1, [208].log_data[16].valid := 1, [208].log_data[17].valid := 1, [208].log_data[18].valid := 1, [208].log_data[19].valid := 1, [208].time.Year := 2023, [208].time.Month := 1, [208].time.Day := 18, [208].time.Hour := 17, [208].time.Minute := 44, [208].time.Second := 59, [209].log_data[0].min := 1.0, [209].log_data[0].max := 1.0, [209].log_data[0].total := 300.0, [209].log_data[0].time := 300.0, [209].log_data[0].minminute := 45, [209].log_data[0].maxminute := 45, [209].log_data[0].valid := 1, [209].log_data[1].valid := 1, [209].log_data[2].valid := 1, [209].log_data[3].valid := 1, [209].log_data[4].valid := 1, [209].log_data[5].valid := 1, [209].log_data[6].valid := 1, [209].log_data[7].valid := 1,
        [209].log_data[8].valid := 1, [209].log_data[9].valid := 1, [209].log_data[10].valid := 1, [209].log_data[11].valid := 1, [209].log_data[12].valid := 1, [209].log_data[13].valid := 1, [209].log_data[14].valid := 1, [209].log_data[15].valid := 1, [209].log_data[16].valid := 1, [209].log_data[17].valid := 1, [209].log_data[18].valid := 1, [209].log_data[19].valid := 1, [209].time.Year := 2023, [209].time.Month := 1, [209].time.Day := 18, [209].time.Hour := 17, [209].time.Minute := 49, [209].time.Second := 59, [210].log_data[0].min := 1.0, [210].log_data[0].max := 1.0, [210].log_data[0].total := 300.0, [210].log_data[0].time := 300.0, [210].log_data[0].minminute := 50, [210].log_data[0].maxminute := 50, [210].log_data[0].valid := 1, [210].log_data[1].valid := 1, [210].log_data[2].valid := 1, [210].log_data[3].valid := 1, [210].log_data[4].valid := 1, [210].log_data[5].valid := 1, [210].log_data[6].valid := 1, [210].log_data[7].valid := 1, [210].log_data[8].valid := 1, [210].log_data[9].valid := 1, [210].log_data[10].valid := 1, [210].log_data[11].valid := 1, [210].log_data[12].valid := 1, [210].log_data[13].valid := 1, [210].log_data[14].valid := 1, [210].log_data[15].valid := 1, [210].log_data[16].valid := 1, [210].log_data[17].valid := 1, [210].log_data[18].valid := 1, [210].log_data[19].valid := 1, [210].time.Year := 2023, [210].time.Month := 1, [210].time.Day := 18, [210].time.Hour := 17, [210].time.Minute := 54, [210].time.Second := 59, [211].log_data[0].min := 1.0, [211].log_data[0].max := 1.0, [211].log_data[0].total := 300.0, [211].log_data[0].time := 300.0, [211].log_data[0].minminute := 55, [211].log_data[0].maxminute := 55, [211].log_data[0].valid := 1, [211].log_data[1].valid := 1, [211].log_data[2].valid := 1, [211].log_data[3].valid := 1,
        [211].log_data[4].valid := 1, [211].log_data[5].valid := 1, [211].log_data[6].valid := 1, [211].log_data[7].valid := 1, [211].log_data[8].valid := 1, [211].log_data[9].valid := 1, [211].log_data[10].valid := 1, [211].log_data[11].valid := 1, [211].log_data[12].valid := 1, [211].log_data[13].valid := 1, [211].log_data[14].valid := 1, [211].log_data[15].valid := 1, [211].log_data[16].valid := 1, [211].log_data[17].valid := 1, [211].log_data[18].valid := 1, [211].log_data[19].valid := 1, [211].time.Year := 2023, [211].time.Month := 1, [211].time.Day := 18, [211].time.Hour := 17, [211].time.Minute := 59, [211].time.Second := 59, [212].log_data[0].min := 1.0, [212].log_data[0].max := 1.0, [212].log_data[0].total := 300.0, [212].log_data[0].time := 300.0, [212].log_data[0].valid := 1, [212].log_data[1].valid := 1, [212].log_data[2].valid := 1, [212].log_data[3].valid := 1, [212].log_data[4].valid := 1, [212].log_data[5].valid := 1, [212].log_data[6].valid := 1, [212].log_data[7].valid := 1, [212].log_data[8].valid := 1, [212].log_data[9].valid := 1, [212].log_data[10].valid := 1, [212].log_data[11].valid := 1, [212].log_data[12].valid := 1, [212].log_data[13].valid := 1, [212].log_data[14].valid := 1, [212].log_data[15].valid := 1, [212].log_data[16].valid := 1, [212].log_data[17].valid := 1, [212].log_data[18].valid := 1, [212].log_data[19].valid := 1, [212].time.Year := 2023, [212].time.Month := 1, [212].time.Day := 18, [212].time.Hour := 18, [212].time.Minute := 4, [212].time.Second := 59, [213].log_data[0].min := 1.0, [213].log_data[0].max := 1.0, [213].log_data[0].total := 300.0, [213].log_data[0].time := 300.0, [213].log_data[0].minminute := 5, [213].log_data[0].maxminute := 5, [213].log_data[0].valid := 1, [213].log_data[1].valid := 1,
        [213].log_data[2].valid := 1, [213].log_data[3].valid := 1, [213].log_data[4].valid := 1, [213].log_data[5].valid := 1, [213].log_data[6].valid := 1, [213].log_data[7].valid := 1, [213].log_data[8].valid := 1, [213].log_data[9].valid := 1, [213].log_data[10].valid := 1, [213].log_data[11].valid := 1, [213].log_data[12].valid := 1, [213].log_data[13].valid := 1, [213].log_data[14].valid := 1, [213].log_data[15].valid := 1, [213].log_data[16].valid := 1, [213].log_data[17].valid := 1, [213].log_data[18].valid := 1, [213].log_data[19].valid := 1, [213].time.Year := 2023, [213].time.Month := 1, [213].time.Day := 18, [213].time.Hour := 18, [213].time.Minute := 9, [213].time.Second := 59, [214].log_data[0].min := 1.0, [214].log_data[0].max := 1.0, [214].log_data[0].total := 300.0, [214].log_data[0].time := 300.0, [214].log_data[0].minminute := 10, [214].log_data[0].maxminute := 10, [214].log_data[0].valid := 1, [214].log_data[1].valid := 1, [214].log_data[2].valid := 1, [214].log_data[3].valid := 1, [214].log_data[4].valid := 1, [214].log_data[5].valid := 1, [214].log_data[6].valid := 1, [214].log_data[7].valid := 1, [214].log_data[8].valid := 1, [214].log_data[9].valid := 1, [214].log_data[10].valid := 1, [214].log_data[11].valid := 1, [214].log_data[12].valid := 1, [214].log_data[13].valid := 1, [214].log_data[14].valid := 1, [214].log_data[15].valid := 1, [214].log_data[16].valid := 1, [214].log_data[17].valid := 1, [214].log_data[18].valid := 1, [214].log_data[19].valid := 1, [214].time.Year := 2023, [214].time.Month := 1, [214].time.Day := 18, [214].time.Hour := 18, [214].time.Minute := 14, [214].time.Second := 59, [215].log_data[0].min := 1.0, [215].log_data[0].max := 1.0, [215].log_data[0].total := 300.0, [215].log_data[0].time := 300.0,
        [215].log_data[0].minminute := 15, [215].log_data[0].maxminute := 15, [215].log_data[0].valid := 1, [215].log_data[1].valid := 1, [215].log_data[2].valid := 1, [215].log_data[3].valid := 1, [215].log_data[4].valid := 1, [215].log_data[5].valid := 1, [215].log_data[6].valid := 1, [215].log_data[7].valid := 1, [215].log_data[8].valid := 1, [215].log_data[9].valid := 1, [215].log_data[10].valid := 1, [215].log_data[11].valid := 1, [215].log_data[12].valid := 1, [215].log_data[13].valid := 1, [215].log_data[14].valid := 1, [215].log_data[15].valid := 1, [215].log_data[16].valid := 1, [215].log_data[17].valid := 1, [215].log_data[18].valid := 1, [215].log_data[19].valid := 1, [215].time.Year := 2023, [215].time.Month := 1, [215].time.Day := 18, [215].time.Hour := 18, [215].time.Minute := 19, [215].time.Second := 59, [216].log_data[0].min := 1.0, [216].log_data[0].max := 1.0, [216].log_data[0].total := 300.0, [216].log_data[0].time := 300.0, [216].log_data[0].minminute := 20, [216].log_data[0].maxminute := 20, [216].log_data[0].valid := 1, [216].log_data[1].valid := 1, [216].log_data[2].valid := 1, [216].log_data[3].valid := 1, [216].log_data[4].valid := 1, [216].log_data[5].valid := 1, [216].log_data[6].valid := 1, [216].log_data[7].valid := 1, [216].log_data[8].valid := 1, [216].log_data[9].valid := 1, [216].log_data[10].valid := 1, [216].log_data[11].valid := 1, [216].log_data[12].valid := 1, [216].log_data[13].valid := 1, [216].log_data[14].valid := 1, [216].log_data[15].valid := 1, [216].log_data[16].valid := 1, [216].log_data[17].valid := 1, [216].log_data[18].valid := 1, [216].log_data[19].valid := 1, [216].time.Year := 2023, [216].time.Month := 1, [216].time.Day := 18, [216].time.Hour := 18, [216].time.Minute := 24, [216].time.Second := 59,
        [217].log_data[0].min := 1.0, [217].log_data[0].max := 1.0, [217].log_data[0].total := 300.0, [217].log_data[0].time := 300.0, [217].log_data[0].minminute := 25, [217].log_data[0].maxminute := 25, [217].log_data[0].valid := 1, [217].log_data[1].valid := 1, [217].log_data[2].valid := 1, [217].log_data[3].valid := 1, [217].log_data[4].valid := 1, [217].log_data[5].valid := 1, [217].log_data[6].valid := 1, [217].log_data[7].valid := 1, [217].log_data[8].valid := 1, [217].log_data[9].valid := 1, [217].log_data[10].valid := 1, [217].log_data[11].valid := 1, [217].log_data[12].valid := 1, [217].log_data[13].valid := 1, [217].log_data[14].valid := 1, [217].log_data[15].valid := 1, [217].log_data[16].valid := 1, [217].log_data[17].valid := 1, [217].log_data[18].valid := 1, [217].log_data[19].valid := 1, [217].time.Year := 2023, [217].time.Month := 1, [217].time.Day := 18, [217].time.Hour := 18, [217].time.Minute := 29, [217].time.Second := 59, [218].log_data[0].min := 1.0, [218].log_data[0].max := 1.0, [218].log_data[0].total := 300.0, [218].log_data[0].time := 300.0, [218].log_data[0].minminute := 30, [218].log_data[0].maxminute := 30, [218].log_data[0].valid := 1, [218].log_data[1].valid := 1, [218].log_data[2].valid := 1, [218].log_data[3].valid := 1, [218].log_data[4].valid := 1, [218].log_data[5].valid := 1, [218].log_data[6].valid := 1, [218].log_data[7].valid := 1, [218].log_data[8].valid := 1, [218].log_data[9].valid := 1, [218].log_data[10].valid := 1, [218].log_data[11].valid := 1, [218].log_data[12].valid := 1, [218].log_data[13].valid := 1, [218].log_data[14].valid := 1, [218].log_data[15].valid := 1, [218].log_data[16].valid := 1, [218].log_data[17].valid := 1, [218].log_data[18].valid := 1, [218].log_data[19].valid := 1, [218].time.Year := 2023, [218].time.Month := 1,
        [218].time.Day := 18, [218].time.Hour := 18, [218].time.Minute := 34, [218].time.Second := 59, [219].log_data[0].min := 1.0, [219].log_data[0].max := 1.0, [219].log_data[0].total := 300.0, [219].log_data[0].time := 300.0, [219].log_data[0].minminute := 35, [219].log_data[0].maxminute := 35, [219].log_data[0].valid := 1, [219].log_data[1].valid := 1, [219].log_data[2].valid := 1, [219].log_data[3].valid := 1, [219].log_data[4].valid := 1, [219].log_data[5].valid := 1, [219].log_data[6].valid := 1, [219].log_data[7].valid := 1, [219].log_data[8].valid := 1, [219].log_data[9].valid := 1, [219].log_data[10].valid := 1, [219].log_data[11].valid := 1, [219].log_data[12].valid := 1, [219].log_data[13].valid := 1, [219].log_data[14].valid := 1, [219].log_data[15].valid := 1, [219].log_data[16].valid := 1, [219].log_data[17].valid := 1, [219].log_data[18].valid := 1, [219].log_data[19].valid := 1, [219].time.Year := 2023, [219].time.Month := 1, [219].time.Day := 18, [219].time.Hour := 18, [219].time.Minute := 39, [219].time.Second := 59, [220].log_data[0].min := 1.0, [220].log_data[0].max := 1.0, [220].log_data[0].total := 300.0, [220].log_data[0].time := 300.0, [220].log_data[0].minminute := 40, [220].log_data[0].maxminute := 40, [220].log_data[0].valid := 1, [220].log_data[1].valid := 1, [220].log_data[2].valid := 1, [220].log_data[3].valid := 1, [220].log_data[4].valid := 1, [220].log_data[5].valid := 1, [220].log_data[6].valid := 1, [220].log_data[7].valid := 1, [220].log_data[8].valid := 1, [220].log_data[9].valid := 1, [220].log_data[10].valid := 1, [220].log_data[11].valid := 1, [220].log_data[12].valid := 1, [220].log_data[13].valid := 1, [220].log_data[14].valid := 1, [220].log_data[15].valid := 1, [220].log_data[16].valid := 1, [220].log_data[17].valid := 1,
        [220].log_data[18].valid := 1, [220].log_data[19].valid := 1, [220].time.Year := 2023, [220].time.Month := 1, [220].time.Day := 18, [220].time.Hour := 18, [220].time.Minute := 44, [220].time.Second := 59, [221].log_data[0].min := 1.0, [221].log_data[0].max := 1.0, [221].log_data[0].total := 300.0, [221].log_data[0].time := 300.0, [221].log_data[0].minminute := 45, [221].log_data[0].maxminute := 45, [221].log_data[0].valid := 1, [221].log_data[1].valid := 1, [221].log_data[2].valid := 1, [221].log_data[3].valid := 1, [221].log_data[4].valid := 1, [221].log_data[5].valid := 1, [221].log_data[6].valid := 1, [221].log_data[7].valid := 1, [221].log_data[8].valid := 1, [221].log_data[9].valid := 1, [221].log_data[10].valid := 1, [221].log_data[11].valid := 1, [221].log_data[12].valid := 1, [221].log_data[13].valid := 1, [221].log_data[14].valid := 1, [221].log_data[15].valid := 1, [221].log_data[16].valid := 1, [221].log_data[17].valid := 1, [221].log_data[18].valid := 1, [221].log_data[19].valid := 1, [221].time.Year := 2023, [221].time.Month := 1, [221].time.Day := 18, [221].time.Hour := 18, [221].time.Minute := 49, [221].time.Second := 59, [222].log_data[0].min := 1.0, [222].log_data[0].max := 1.0, [222].log_data[0].total := 300.0, [222].log_data[0].time := 300.0, [222].log_data[0].minminute := 50, [222].log_data[0].maxminute := 50, [222].log_data[0].valid := 1, [222].log_data[1].valid := 1, [222].log_data[2].valid := 1, [222].log_data[3].valid := 1, [222].log_data[4].valid := 1, [222].log_data[5].valid := 1, [222].log_data[6].valid := 1, [222].log_data[7].valid := 1, [222].log_data[8].valid := 1, [222].log_data[9].valid := 1, [222].log_data[10].valid := 1, [222].log_data[11].valid := 1, [222].log_data[12].valid := 1, [222].log_data[13].valid := 1,
        [222].log_data[14].valid := 1, [222].log_data[15].valid := 1, [222].log_data[16].valid := 1, [222].log_data[17].valid := 1, [222].log_data[18].valid := 1, [222].log_data[19].valid := 1, [222].time.Year := 2023, [222].time.Month := 1, [222].time.Day := 18, [222].time.Hour := 18, [222].time.Minute := 54, [222].time.Second := 59, [223].log_data[0].min := 1.0, [223].log_data[0].max := 1.0, [223].log_data[0].total := 300.0, [223].log_data[0].time := 300.0, [223].log_data[0].minminute := 55, [223].log_data[0].maxminute := 55, [223].log_data[0].valid := 1, [223].log_data[1].valid := 1, [223].log_data[2].valid := 1, [223].log_data[3].valid := 1, [223].log_data[4].valid := 1, [223].log_data[5].valid := 1, [223].log_data[6].valid := 1, [223].log_data[7].valid := 1, [223].log_data[8].valid := 1, [223].log_data[9].valid := 1, [223].log_data[10].valid := 1, [223].log_data[11].valid := 1, [223].log_data[12].valid := 1, [223].log_data[13].valid := 1, [223].log_data[14].valid := 1, [223].log_data[15].valid := 1, [223].log_data[16].valid := 1, [223].log_data[17].valid := 1, [223].log_data[18].valid := 1, [223].log_data[19].valid := 1, [223].time.Year := 2023, [223].time.Month := 1, [223].time.Day := 18, [223].time.Hour := 18, [223].time.Minute := 59, [223].time.Second := 59, [224].log_data[0].min := 1.0, [224].log_data[0].max := 1.0, [224].log_data[0].total := 300.0, [224].log_data[0].time := 300.0, [224].log_data[0].valid := 1, [224].log_data[1].valid := 1, [224].log_data[2].valid := 1, [224].log_data[3].valid := 1, [224].log_data[4].valid := 1, [224].log_data[5].valid := 1, [224].log_data[6].valid := 1, [224].log_data[7].valid := 1, [224].log_data[8].valid := 1, [224].log_data[9].valid := 1, [224].log_data[10].valid := 1, [224].log_data[11].valid := 1,
        [224].log_data[12].valid := 1, [224].log_data[13].valid := 1, [224].log_data[14].valid := 1, [224].log_data[15].valid := 1, [224].log_data[16].valid := 1, [224].log_data[17].valid := 1, [224].log_data[18].valid := 1, [224].log_data[19].valid := 1, [224].time.Year := 2023, [224].time.Month := 1, [224].time.Day := 18, [224].time.Hour := 19, [224].time.Minute := 4, [224].time.Second := 59, [225].log_data[0].min := 1.0, [225].log_data[0].max := 1.0, [225].log_data[0].total := 300.0, [225].log_data[0].time := 300.0, [225].log_data[0].minminute := 5, [225].log_data[0].maxminute := 5, [225].log_data[0].valid := 1, [225].log_data[1].valid := 1, [225].log_data[2].valid := 1, [225].log_data[3].valid := 1, [225].log_data[4].valid := 1, [225].log_data[5].valid := 1, [225].log_data[6].valid := 1, [225].log_data[7].valid := 1, [225].log_data[8].valid := 1, [225].log_data[9].valid := 1, [225].log_data[10].valid := 1, [225].log_data[11].valid := 1, [225].log_data[12].valid := 1, [225].log_data[13].valid := 1, [225].log_data[14].valid := 1, [225].log_data[15].valid := 1, [225].log_data[16].valid := 1, [225].log_data[17].valid := 1, [225].log_data[18].valid := 1, [225].log_data[19].valid := 1, [225].time.Year := 2023, [225].time.Month := 1, [225].time.Day := 18, [225].time.Hour := 19, [225].time.Minute := 9, [225].time.Second := 59, [226].log_data[0].min := 1.0, [226].log_data[0].max := 1.0, [226].log_data[0].total := 300.0, [226].log_data[0].time := 300.0, [226].log_data[0].minminute := 10, [226].log_data[0].maxminute := 10, [226].log_data[0].valid := 1, [226].log_data[1].valid := 1, [226].log_data[2].valid := 1, [226].log_data[3].valid := 1, [226].log_data[4].valid := 1, [226].log_data[5].valid := 1, [226].log_data[6].valid := 1, [226].log_data[7].valid := 1,
        [226].log_data[8].valid := 1, [226].log_data[9].valid := 1, [226].log_data[10].valid := 1, [226].log_data[11].valid := 1, [226].log_data[12].valid := 1, [226].log_data[13].valid := 1, [226].log_data[14].valid := 1, [226].log_data[15].valid := 1, [226].log_data[16].valid := 1, [226].log_data[17].valid := 1, [226].log_data[18].valid := 1, [226].log_data[19].valid := 1, [226].time.Year := 2023, [226].time.Month := 1, [226].time.Day := 18, [226].time.Hour := 19, [226].time.Minute := 14, [226].time.Second := 59, [227].log_data[0].min := 1.0, [227].log_data[0].max := 1.0, [227].log_data[0].total := 300.0, [227].log_data[0].time := 300.0, [227].log_data[0].minminute := 15, [227].log_data[0].maxminute := 15, [227].log_data[0].valid := 1, [227].log_data[1].valid := 1, [227].log_data[2].valid := 1, [227].log_data[3].valid := 1, [227].log_data[4].valid := 1, [227].log_data[5].valid := 1, [227].log_data[6].valid := 1, [227].log_data[7].valid := 1, [227].log_data[8].valid := 1, [227].log_data[9].valid := 1, [227].log_data[10].valid := 1, [227].log_data[11].valid := 1, [227].log_data[12].valid := 1, [227].log_data[13].valid := 1, [227].log_data[14].valid := 1, [227].log_data[15].valid := 1, [227].log_data[16].valid := 1, [227].log_data[17].valid := 1, [227].log_data[18].valid := 1, [227].log_data[19].valid := 1, [227].time.Year := 2023, [227].time.Month := 1, [227].time.Day := 18, [227].time.Hour := 19, [227].time.Minute := 19, [227].time.Second := 59, [228].log_data[0].min := 1.0, [228].log_data[0].max := 1.0, [228].log_data[0].total := 300.0, [228].log_data[0].time := 300.0, [228].log_data[0].minminute := 20, [228].log_data[0].maxminute := 20, [228].log_data[0].valid := 1, [228].log_data[1].valid := 1, [228].log_data[2].valid := 1, [228].log_data[3].valid := 1,
        [228].log_data[4].valid := 1, [228].log_data[5].valid := 1, [228].log_data[6].valid := 1, [228].log_data[7].valid := 1, [228].log_data[8].valid := 1, [228].log_data[9].valid := 1, [228].log_data[10].valid := 1, [228].log_data[11].valid := 1, [228].log_data[12].valid := 1, [228].log_data[13].valid := 1, [228].log_data[14].valid := 1, [228].log_data[15].valid := 1, [228].log_data[16].valid := 1, [228].log_data[17].valid := 1, [228].log_data[18].valid := 1, [228].log_data[19].valid := 1, [228].time.Year := 2023, [228].time.Month := 1, [228].time.Day := 18, [228].time.Hour := 19, [228].time.Minute := 24, [228].time.Second := 59, [229].log_data[0].min := 1.0, [229].log_data[0].max := 1.0, [229].log_data[0].total := 300.0, [229].log_data[0].time := 300.0, [229].log_data[0].minminute := 25, [229].log_data[0].maxminute := 25, [229].log_data[0].valid := 1, [229].log_data[1].valid := 1, [229].log_data[2].valid := 1, [229].log_data[3].valid := 1, [229].log_data[4].valid := 1, [229].log_data[5].valid := 1, [229].log_data[6].valid := 1, [229].log_data[7].valid := 1, [229].log_data[8].valid := 1, [229].log_data[9].valid := 1, [229].log_data[10].valid := 1, [229].log_data[11].valid := 1, [229].log_data[12].valid := 1, [229].log_data[13].valid := 1, [229].log_data[14].valid := 1, [229].log_data[15].valid := 1, [229].log_data[16].valid := 1, [229].log_data[17].valid := 1, [229].log_data[18].valid := 1, [229].log_data[19].valid := 1, [229].time.Year := 2023, [229].time.Month := 1, [229].time.Day := 18, [229].time.Hour := 19, [229].time.Minute := 29, [229].time.Second := 59, [230].log_data[0].min := 1.0, [230].log_data[0].max := 1.0, [230].log_data[0].total := 300.0, [230].log_data[0].time := 300.0, [230].log_data[0].minminute := 30, [230].log_data[0].maxminute := 30,
        [230].log_data[0].valid := 1, [230].log_data[1].valid := 1, [230].log_data[2].valid := 1, [230].log_data[3].valid := 1, [230].log_data[4].valid := 1, [230].log_data[5].valid := 1, [230].log_data[6].valid := 1, [230].log_data[7].valid := 1, [230].log_data[8].valid := 1, [230].log_data[9].valid := 1, [230].log_data[10].valid := 1, [230].log_data[11].valid := 1, [230].log_data[12].valid := 1, [230].log_data[13].valid := 1, [230].log_data[14].valid := 1, [230].log_data[15].valid := 1, [230].log_data[16].valid := 1, [230].log_data[17].valid := 1, [230].log_data[18].valid := 1, [230].log_data[19].valid := 1, [230].time.Year := 2023, [230].time.Month := 1, [230].time.Day := 18, [230].time.Hour := 19, [230].time.Minute := 34, [230].time.Second := 59, [231].log_data[0].min := 1.0, [231].log_data[0].max := 1.0, [231].log_data[0].total := 300.0, [231].log_data[0].time := 300.0, [231].log_data[0].minminute := 35, [231].log_data[0].maxminute := 35, [231].log_data[0].valid := 1, [231].log_data[1].valid := 1, [231].log_data[2].valid := 1, [231].log_data[3].valid := 1, [231].log_data[4].valid := 1, [231].log_data[5].valid := 1, [231].log_data[6].valid := 1, [231].log_data[7].valid := 1, [231].log_data[8].valid := 1, [231].log_data[9].valid := 1, [231].log_data[10].valid := 1, [231].log_data[11].valid := 1, [231].log_data[12].valid := 1, [231].log_data[13].valid := 1, [231].log_data[14].valid := 1, [231].log_data[15].valid := 1, [231].log_data[16].valid := 1, [231].log_data[17].valid := 1, [231].log_data[18].valid := 1, [231].log_data[19].valid := 1, [231].time.Year := 2023, [231].time.Month := 1, [231].time.Day := 18, [231].time.Hour := 19, [231].time.Minute := 39, [231].time.Second := 59, [232].log_data[0].min := 1.0, [232].log_data[0].max := 1.0,
        [232].log_data[0].total := 300.0, [232].log_data[0].time := 300.0, [232].log_data[0].minminute := 40, [232].log_data[0].maxminute := 40, [232].log_data[0].valid := 1, [232].log_data[1].valid := 1, [232].log_data[2].valid := 1, [232].log_data[3].valid := 1, [232].log_data[4].valid := 1, [232].log_data[5].valid := 1, [232].log_data[6].valid := 1, [232].log_data[7].valid := 1, [232].log_data[8].valid := 1, [232].log_data[9].valid := 1, [232].log_data[10].valid := 1, [232].log_data[11].valid := 1, [232].log_data[12].valid := 1, [232].log_data[13].valid := 1, [232].log_data[14].valid := 1, [232].log_data[15].valid := 1, [232].log_data[16].valid := 1, [232].log_data[17].valid := 1, [232].log_data[18].valid := 1, [232].log_data[19].valid := 1, [232].time.Year := 2023, [232].time.Month := 1, [232].time.Day := 18, [232].time.Hour := 19, [232].time.Minute := 44, [232].time.Second := 59, [233].log_data[0].min := 1.0, [233].log_data[0].max := 1.0, [233].log_data[0].total := 300.0, [233].log_data[0].time := 300.0, [233].log_data[0].minminute := 45, [233].log_data[0].maxminute := 45, [233].log_data[0].valid := 1, [233].log_data[1].valid := 1, [233].log_data[2].valid := 1, [233].log_data[3].valid := 1, [233].log_data[4].valid := 1, [233].log_data[5].valid := 1, [233].log_data[6].valid := 1, [233].log_data[7].valid := 1, [233].log_data[8].valid := 1, [233].log_data[9].valid := 1, [233].log_data[10].valid := 1, [233].log_data[11].valid := 1, [233].log_data[12].valid := 1, [233].log_data[13].valid := 1, [233].log_data[14].valid := 1, [233].log_data[15].valid := 1, [233].log_data[16].valid := 1, [233].log_data[17].valid := 1, [233].log_data[18].valid := 1, [233].log_data[19].valid := 1, [233].time.Year := 2023, [233].time.Month := 1, [233].time.Day := 18, [233].time.Hour := 19,
        [233].time.Minute := 49, [233].time.Second := 59, [234].log_data[0].min := 1.0, [234].log_data[0].max := 1.0, [234].log_data[0].total := 300.0, [234].log_data[0].time := 300.0, [234].log_data[0].minminute := 50, [234].log_data[0].maxminute := 50, [234].log_data[0].valid := 1, [234].log_data[1].valid := 1, [234].log_data[2].valid := 1, [234].log_data[3].valid := 1, [234].log_data[4].valid := 1, [234].log_data[5].valid := 1, [234].log_data[6].valid := 1, [234].log_data[7].valid := 1, [234].log_data[8].valid := 1, [234].log_data[9].valid := 1, [234].log_data[10].valid := 1, [234].log_data[11].valid := 1, [234].log_data[12].valid := 1, [234].log_data[13].valid := 1, [234].log_data[14].valid := 1, [234].log_data[15].valid := 1, [234].log_data[16].valid := 1, [234].log_data[17].valid := 1, [234].log_data[18].valid := 1, [234].log_data[19].valid := 1, [234].time.Year := 2023, [234].time.Month := 1, [234].time.Day := 18, [234].time.Hour := 19, [234].time.Minute := 54, [234].time.Second := 59, [235].log_data[0].min := 1.0, [235].log_data[0].max := 1.0, [235].log_data[0].total := 300.0, [235].log_data[0].time := 300.0, [235].log_data[0].minminute := 55, [235].log_data[0].maxminute := 55, [235].log_data[0].valid := 1, [235].log_data[1].valid := 1, [235].log_data[2].valid := 1, [235].log_data[3].valid := 1, [235].log_data[4].valid := 1, [235].log_data[5].valid := 1, [235].log_data[6].valid := 1, [235].log_data[7].valid := 1, [235].log_data[8].valid := 1, [235].log_data[9].valid := 1, [235].log_data[10].valid := 1, [235].log_data[11].valid := 1, [235].log_data[12].valid := 1, [235].log_data[13].valid := 1, [235].log_data[14].valid := 1, [235].log_data[15].valid := 1, [235].log_data[16].valid := 1, [235].log_data[17].valid := 1, [235].log_data[18].valid := 1, [235].log_data[19].valid := 1,
        [235].time.Year := 2023, [235].time.Month := 1, [235].time.Day := 18, [235].time.Hour := 19, [235].time.Minute := 59, [235].time.Second := 59, [236].log_data[0].min := 1.0, [236].log_data[0].max := 1.0, [236].log_data[0].total := 300.0, [236].log_data[0].time := 300.0, [236].log_data[0].valid := 1, [236].log_data[1].valid := 1, [236].log_data[2].valid := 1, [236].log_data[3].valid := 1, [236].log_data[4].valid := 1, [236].log_data[5].valid := 1, [236].log_data[6].valid := 1, [236].log_data[7].valid := 1, [236].log_data[8].valid := 1, [236].log_data[9].valid := 1, [236].log_data[10].valid := 1, [236].log_data[11].valid := 1, [236].log_data[12].valid := 1, [236].log_data[13].valid := 1, [236].log_data[14].valid := 1, [236].log_data[15].valid := 1, [236].log_data[16].valid := 1, [236].log_data[17].valid := 1, [236].log_data[18].valid := 1, [236].log_data[19].valid := 1, [236].time.Year := 2023, [236].time.Month := 1, [236].time.Day := 18, [236].time.Hour := 20, [236].time.Minute := 4, [236].time.Second := 59, [237].log_data[0].min := 1.0, [237].log_data[0].max := 1.0, [237].log_data[0].total := 300.0, [237].log_data[0].time := 300.0, [237].log_data[0].minminute := 5, [237].log_data[0].maxminute := 5, [237].log_data[0].valid := 1, [237].log_data[1].valid := 1, [237].log_data[2].valid := 1, [237].log_data[3].valid := 1, [237].log_data[4].valid := 1, [237].log_data[5].valid := 1, [237].log_data[6].valid := 1, [237].log_data[7].valid := 1, [237].log_data[8].valid := 1, [237].log_data[9].valid := 1, [237].log_data[10].valid := 1, [237].log_data[11].valid := 1, [237].log_data[12].valid := 1, [237].log_data[13].valid := 1, [237].log_data[14].valid := 1, [237].log_data[15].valid := 1, [237].log_data[16].valid := 1, [237].log_data[17].valid := 1,
        [237].log_data[18].valid := 1, [237].log_data[19].valid := 1, [237].time.Year := 2023, [237].time.Month := 1, [237].time.Day := 18, [237].time.Hour := 20, [237].time.Minute := 9, [237].time.Second := 59, [238].log_data[0].min := 1.0, [238].log_data[0].max := 1.0, [238].log_data[0].total := 300.0, [238].log_data[0].time := 300.0, [238].log_data[0].minminute := 10, [238].log_data[0].maxminute := 10, [238].log_data[0].valid := 1, [238].log_data[1].valid := 1, [238].log_data[2].valid := 1, [238].log_data[3].valid := 1, [238].log_data[4].valid := 1, [238].log_data[5].valid := 1, [238].log_data[6].valid := 1, [238].log_data[7].valid := 1, [238].log_data[8].valid := 1, [238].log_data[9].valid := 1, [238].log_data[10].valid := 1, [238].log_data[11].valid := 1, [238].log_data[12].valid := 1, [238].log_data[13].valid := 1, [238].log_data[14].valid := 1, [238].log_data[15].valid := 1, [238].log_data[16].valid := 1, [238].log_data[17].valid := 1, [238].log_data[18].valid := 1, [238].log_data[19].valid := 1, [238].time.Year := 2023, [238].time.Month := 1, [238].time.Day := 18, [238].time.Hour := 20, [238].time.Minute := 14, [238].time.Second := 59, [239].log_data[0].min := 1.0, [239].log_data[0].max := 1.0, [239].log_data[0].total := 300.0, [239].log_data[0].time := 300.0, [239].log_data[0].minminute := 15, [239].log_data[0].maxminute := 15, [239].log_data[0].valid := 1, [239].log_data[1].valid := 1, [239].log_data[2].valid := 1, [239].log_data[3].valid := 1, [239].log_data[4].valid := 1, [239].log_data[5].valid := 1, [239].log_data[6].valid := 1, [239].log_data[7].valid := 1, [239].log_data[8].valid := 1, [239].log_data[9].valid := 1, [239].log_data[10].valid := 1, [239].log_data[11].valid := 1, [239].log_data[12].valid := 1, [239].log_data[13].valid := 1,
        [239].log_data[14].valid := 1, [239].log_data[15].valid := 1, [239].log_data[16].valid := 1, [239].log_data[17].valid := 1, [239].log_data[18].valid := 1, [239].log_data[19].valid := 1, [239].time.Year := 2023, [239].time.Month := 1, [239].time.Day := 18, [239].time.Hour := 20, [239].time.Minute := 19, [239].time.Second := 59, [240].log_data[0].min := 1.0, [240].log_data[0].max := 1.0, [240].log_data[0].total := 300.0, [240].log_data[0].time := 300.0, [240].log_data[0].minminute := 20, [240].log_data[0].maxminute := 20, [240].log_data[0].valid := 1, [240].log_data[1].valid := 1, [240].log_data[2].valid := 1, [240].log_data[3].valid := 1, [240].log_data[4].valid := 1, [240].log_data[5].valid := 1, [240].log_data[6].valid := 1, [240].log_data[7].valid := 1, [240].log_data[8].valid := 1, [240].log_data[9].valid := 1, [240].log_data[10].valid := 1, [240].log_data[11].valid := 1, [240].log_data[12].valid := 1, [240].log_data[13].valid := 1, [240].log_data[14].valid := 1, [240].log_data[15].valid := 1, [240].log_data[16].valid := 1, [240].log_data[17].valid := 1, [240].log_data[18].valid := 1, [240].log_data[19].valid := 1, [240].time.Year := 2023, [240].time.Month := 1, [240].time.Day := 18, [240].time.Hour := 20, [240].time.Minute := 24, [240].time.Second := 59, [241].log_data[0].min := 1.0, [241].log_data[0].max := 1.0, [241].log_data[0].total := 300.0, [241].log_data[0].time := 300.0, [241].log_data[0].minminute := 25, [241].log_data[0].maxminute := 25, [241].log_data[0].valid := 1, [241].log_data[1].valid := 1, [241].log_data[2].valid := 1, [241].log_data[3].valid := 1, [241].log_data[4].valid := 1, [241].log_data[5].valid := 1, [241].log_data[6].valid := 1, [241].log_data[7].valid := 1, [241].log_data[8].valid := 1, [241].log_data[9].valid := 1,
        [241].log_data[10].valid := 1, [241].log_data[11].valid := 1, [241].log_data[12].valid := 1, [241].log_data[13].valid := 1, [241].log_data[14].valid := 1, [241].log_data[15].valid := 1, [241].log_data[16].valid := 1, [241].log_data[17].valid := 1, [241].log_data[18].valid := 1, [241].log_data[19].valid := 1, [241].time.Year := 2023, [241].time.Month := 1, [241].time.Day := 18, [241].time.Hour := 20, [241].time.Minute := 29, [241].time.Second := 59, [242].log_data[0].min := 1.0, [242].log_data[0].max := 1.0, [242].log_data[0].total := 300.0, [242].log_data[0].time := 300.0, [242].log_data[0].minminute := 30, [242].log_data[0].maxminute := 30, [242].log_data[0].valid := 1, [242].log_data[1].valid := 1, [242].log_data[2].valid := 1, [242].log_data[3].valid := 1, [242].log_data[4].valid := 1, [242].log_data[5].valid := 1, [242].log_data[6].valid := 1, [242].log_data[7].valid := 1, [242].log_data[8].valid := 1, [242].log_data[9].valid := 1, [242].log_data[10].valid := 1, [242].log_data[11].valid := 1, [242].log_data[12].valid := 1, [242].log_data[13].valid := 1, [242].log_data[14].valid := 1, [242].log_data[15].valid := 1, [242].log_data[16].valid := 1, [242].log_data[17].valid := 1, [242].log_data[18].valid := 1, [242].log_data[19].valid := 1, [242].time.Year := 2023, [242].time.Month := 1, [242].time.Day := 18, [242].time.Hour := 20, [242].time.Minute := 34, [242].time.Second := 59, [243].log_data[0].min := 1.0, [243].log_data[0].max := 1.0, [243].log_data[0].total := 300.0, [243].log_data[0].time := 300.0, [243].log_data[0].minminute := 35, [243].log_data[0].maxminute := 35, [243].log_data[0].valid := 1, [243].log_data[1].valid := 1, [243].log_data[2].valid := 1, [243].log_data[3].valid := 1, [243].log_data[4].valid := 1, [243].log_data[5].valid := 1,
        [243].log_data[6].valid := 1, [243].log_data[7].valid := 1, [243].log_data[8].valid := 1, [243].log_data[9].valid := 1, [243].log_data[10].valid := 1, [243].log_data[11].valid := 1, [243].log_data[12].valid := 1, [243].log_data[13].valid := 1, [243].log_data[14].valid := 1, [243].log_data[15].valid := 1, [243].log_data[16].valid := 1, [243].log_data[17].valid := 1, [243].log_data[18].valid := 1, [243].log_data[19].valid := 1, [243].time.Year := 2023, [243].time.Month := 1, [243].time.Day := 18, [243].time.Hour := 20, [243].time.Minute := 39, [243].time.Second := 59, [244].log_data[0].min := 1.0, [244].log_data[0].max := 1.0, [244].log_data[0].total := 300.0, [244].log_data[0].time := 300.0, [244].log_data[0].minminute := 40, [244].log_data[0].maxminute := 40, [244].log_data[0].valid := 1, [244].log_data[1].valid := 1, [244].log_data[2].valid := 1, [244].log_data[3].valid := 1, [244].log_data[4].valid := 1, [244].log_data[5].valid := 1, [244].log_data[6].valid := 1, [244].log_data[7].valid := 1, [244].log_data[8].valid := 1, [244].log_data[9].valid := 1, [244].log_data[10].valid := 1, [244].log_data[11].valid := 1, [244].log_data[12].valid := 1, [244].log_data[13].valid := 1, [244].log_data[14].valid := 1, [244].log_data[15].valid := 1, [244].log_data[16].valid := 1, [244].log_data[17].valid := 1, [244].log_data[18].valid := 1, [244].log_data[19].valid := 1, [244].time.Year := 2023, [244].time.Month := 1, [244].time.Day := 18, [244].time.Hour := 20, [244].time.Minute := 44, [244].time.Second := 59, [245].log_data[0].min := 1.0, [245].log_data[0].max := 1.0, [245].log_data[0].total := 300.0, [245].log_data[0].time := 300.0, [245].log_data[0].minminute := 45, [245].log_data[0].maxminute := 45, [245].log_data[0].valid := 1, [245].log_data[1].valid := 1,
        [245].log_data[2].valid := 1, [245].log_data[3].valid := 1, [245].log_data[4].valid := 1, [245].log_data[5].valid := 1, [245].log_data[6].valid := 1, [245].log_data[7].valid := 1, [245].log_data[8].valid := 1, [245].log_data[9].valid := 1, [245].log_data[10].valid := 1, [245].log_data[11].valid := 1, [245].log_data[12].valid := 1, [245].log_data[13].valid := 1, [245].log_data[14].valid := 1, [245].log_data[15].valid := 1, [245].log_data[16].valid := 1, [245].log_data[17].valid := 1, [245].log_data[18].valid := 1, [245].log_data[19].valid := 1, [245].time.Year := 2023, [245].time.Month := 1, [245].time.Day := 18, [245].time.Hour := 20, [245].time.Minute := 49, [245].time.Second := 59, [246].log_data[0].min := 1.0, [246].log_data[0].max := 1.0, [246].log_data[0].total := 300.0, [246].log_data[0].time := 300.0, [246].log_data[0].minminute := 50, [246].log_data[0].maxminute := 50, [246].log_data[0].valid := 1, [246].log_data[1].valid := 1, [246].log_data[2].valid := 1, [246].log_data[3].valid := 1, [246].log_data[4].valid := 1, [246].log_data[5].valid := 1, [246].log_data[6].valid := 1, [246].log_data[7].valid := 1, [246].log_data[8].valid := 1, [246].log_data[9].valid := 1, [246].log_data[10].valid := 1, [246].log_data[11].valid := 1, [246].log_data[12].valid := 1, [246].log_data[13].valid := 1, [246].log_data[14].valid := 1, [246].log_data[15].valid := 1, [246].log_data[16].valid := 1, [246].log_data[17].valid := 1, [246].log_data[18].valid := 1, [246].log_data[19].valid := 1, [246].time.Year := 2023, [246].time.Month := 1, [246].time.Day := 18, [246].time.Hour := 20, [246].time.Minute := 54, [246].time.Second := 59, [247].log_data[0].min := 1.0, [247].log_data[0].max := 1.0, [247].log_data[0].total := 300.0, [247].log_data[0].time := 300.0,
        [247].log_data[0].minminute := 55, [247].log_data[0].maxminute := 55, [247].log_data[0].valid := 1, [247].log_data[1].valid := 1, [247].log_data[2].valid := 1, [247].log_data[3].valid := 1, [247].log_data[4].valid := 1, [247].log_data[5].valid := 1, [247].log_data[6].valid := 1, [247].log_data[7].valid := 1, [247].log_data[8].valid := 1, [247].log_data[9].valid := 1, [247].log_data[10].valid := 1, [247].log_data[11].valid := 1, [247].log_data[12].valid := 1, [247].log_data[13].valid := 1, [247].log_data[14].valid := 1, [247].log_data[15].valid := 1, [247].log_data[16].valid := 1, [247].log_data[17].valid := 1, [247].log_data[18].valid := 1, [247].log_data[19].valid := 1, [247].time.Year := 2023, [247].time.Month := 1, [247].time.Day := 18, [247].time.Hour := 20, [247].time.Minute := 59, [247].time.Second := 59, [248].log_data[0].min := 1.0, [248].log_data[0].max := 1.0, [248].log_data[0].total := 299.5, [248].log_data[0].time := 299.5, [248].log_data[0].valid := 1, [248].log_data[1].valid := 1, [248].log_data[2].valid := 1, [248].log_data[3].valid := 1, [248].log_data[4].valid := 1, [248].log_data[5].valid := 1, [248].log_data[6].valid := 1, [248].log_data[7].valid := 1, [248].log_data[8].valid := 1, [248].log_data[9].valid := 1, [248].log_data[10].valid := 1, [248].log_data[11].valid := 1, [248].log_data[12].valid := 1, [248].log_data[13].valid := 1, [248].log_data[14].valid := 1, [248].log_data[15].valid := 1, [248].log_data[16].valid := 1, [248].log_data[17].valid := 1, [248].log_data[18].valid := 1, [248].log_data[19].valid := 1, [248].time.Year := 2023, [248].time.Month := 1, [248].time.Day := 18, [248].time.Hour := 21, [248].time.Minute := 4, [248].time.Second := 59, [249].log_data[0].min := 1.0, [249].log_data[0].max := 1.0,
        [249].log_data[0].total := 300.0, [249].log_data[0].time := 300.0, [249].log_data[0].minminute := 5, [249].log_data[0].maxminute := 5, [249].log_data[0].valid := 1, [249].log_data[1].valid := 1, [249].log_data[2].valid := 1, [249].log_data[3].valid := 1, [249].log_data[4].valid := 1, [249].log_data[5].valid := 1, [249].log_data[6].valid := 1, [249].log_data[7].valid := 1, [249].log_data[8].valid := 1, [249].log_data[9].valid := 1, [249].log_data[10].valid := 1, [249].log_data[11].valid := 1, [249].log_data[12].valid := 1, [249].log_data[13].valid := 1, [249].log_data[14].valid := 1, [249].log_data[15].valid := 1, [249].log_data[16].valid := 1, [249].log_data[17].valid := 1, [249].log_data[18].valid := 1, [249].log_data[19].valid := 1, [249].time.Year := 2023, [249].time.Month := 1, [249].time.Day := 18, [249].time.Hour := 21, [249].time.Minute := 9, [249].time.Second := 59, [250].log_data[0].min := 1.0, [250].log_data[0].max := 1.0, [250].log_data[0].total := 300.0, [250].log_data[0].time := 300.0, [250].log_data[0].minminute := 10, [250].log_data[0].maxminute := 10, [250].log_data[0].valid := 1, [250].log_data[1].valid := 1, [250].log_data[2].valid := 1, [250].log_data[3].valid := 1, [250].log_data[4].valid := 1, [250].log_data[5].valid := 1, [250].log_data[6].valid := 1, [250].log_data[7].valid := 1, [250].log_data[8].valid := 1, [250].log_data[9].valid := 1, [250].log_data[10].valid := 1, [250].log_data[11].valid := 1, [250].log_data[12].valid := 1, [250].log_data[13].valid := 1, [250].log_data[14].valid := 1, [250].log_data[15].valid := 1, [250].log_data[16].valid := 1, [250].log_data[17].valid := 1, [250].log_data[18].valid := 1, [250].log_data[19].valid := 1, [250].time.Year := 2023, [250].time.Month := 1, [250].time.Day := 18, [250].time.Hour := 21,
        [250].time.Minute := 14, [250].time.Second := 59, [251].log_data[0].min := 1.0, [251].log_data[0].max := 1.0, [251].log_data[0].total := 300.0, [251].log_data[0].time := 300.0, [251].log_data[0].minminute := 15, [251].log_data[0].maxminute := 15, [251].log_data[0].valid := 1, [251].log_data[1].valid := 1, [251].log_data[2].valid := 1, [251].log_data[3].valid := 1, [251].log_data[4].valid := 1, [251].log_data[5].valid := 1, [251].log_data[6].valid := 1, [251].log_data[7].valid := 1, [251].log_data[8].valid := 1, [251].log_data[9].valid := 1, [251].log_data[10].valid := 1, [251].log_data[11].valid := 1, [251].log_data[12].valid := 1, [251].log_data[13].valid := 1, [251].log_data[14].valid := 1, [251].log_data[15].valid := 1, [251].log_data[16].valid := 1, [251].log_data[17].valid := 1, [251].log_data[18].valid := 1, [251].log_data[19].valid := 1, [251].time.Year := 2023, [251].time.Month := 1, [251].time.Day := 18, [251].time.Hour := 21, [251].time.Minute := 19, [251].time.Second := 59, [252].log_data[0].min := 1.0, [252].log_data[0].max := 1.0, [252].log_data[0].total := 300.0, [252].log_data[0].time := 300.0, [252].log_data[0].minminute := 20, [252].log_data[0].maxminute := 20, [252].log_data[0].valid := 1, [252].log_data[1].valid := 1, [252].log_data[2].valid := 1, [252].log_data[3].valid := 1, [252].log_data[4].valid := 1, [252].log_data[5].valid := 1, [252].log_data[6].valid := 1, [252].log_data[7].valid := 1, [252].log_data[8].valid := 1, [252].log_data[9].valid := 1, [252].log_data[10].valid := 1, [252].log_data[11].valid := 1, [252].log_data[12].valid := 1, [252].log_data[13].valid := 1, [252].log_data[14].valid := 1, [252].log_data[15].valid := 1, [252].log_data[16].valid := 1, [252].log_data[17].valid := 1, [252].log_data[18].valid := 1, [252].log_data[19].valid := 1,
        [252].time.Year := 2023, [252].time.Month := 1, [252].time.Day := 18, [252].time.Hour := 21, [252].time.Minute := 24, [252].time.Second := 59, [253].log_data[0].min := 1.0, [253].log_data[0].max := 1.0, [253].log_data[0].total := 300.0, [253].log_data[0].time := 300.0, [253].log_data[0].minminute := 25, [253].log_data[0].maxminute := 25, [253].log_data[0].valid := 1, [253].log_data[1].valid := 1, [253].log_data[2].valid := 1, [253].log_data[3].valid := 1, [253].log_data[4].valid := 1, [253].log_data[5].valid := 1, [253].log_data[6].valid := 1, [253].log_data[7].valid := 1, [253].log_data[8].valid := 1, [253].log_data[9].valid := 1, [253].log_data[10].valid := 1, [253].log_data[11].valid := 1, [253].log_data[12].valid := 1, [253].log_data[13].valid := 1, [253].log_data[14].valid := 1, [253].log_data[15].valid := 1, [253].log_data[16].valid := 1, [253].log_data[17].valid := 1, [253].log_data[18].valid := 1, [253].log_data[19].valid := 1, [253].time.Year := 2023, [253].time.Month := 1, [253].time.Day := 18, [253].time.Hour := 21, [253].time.Minute := 29, [253].time.Second := 59, [254].log_data[0].min := 1.0, [254].log_data[0].max := 1.0, [254].log_data[0].total := 300.0, [254].log_data[0].time := 300.0, [254].log_data[0].minminute := 30, [254].log_data[0].maxminute := 30, [254].log_data[0].valid := 1, [254].log_data[1].valid := 1, [254].log_data[2].valid := 1, [254].log_data[3].valid := 1, [254].log_data[4].valid := 1, [254].log_data[5].valid := 1, [254].log_data[6].valid := 1, [254].log_data[7].valid := 1, [254].log_data[8].valid := 1, [254].log_data[9].valid := 1, [254].log_data[10].valid := 1, [254].log_data[11].valid := 1, [254].log_data[12].valid := 1, [254].log_data[13].valid := 1, [254].log_data[14].valid := 1, [254].log_data[15].valid := 1,
